// TIA Portal V18 program export: 1 tag tables, 0 data types, 4 data blocks, 6 code blocks (in call order from the OBs), 0 instance data blocks

VAR_GLOBAL   // PLC tag table "AI_Tags"
   AI_Nut_Khoi_Dong AT %I0.0 : Bool;   // Nút khởi động vật lý
   AI_Nut_Khoi_Dong_HMI AT %M110.0 : Bool;   // Tín hiệu mô phỏng/HMI song song cho Nút khởi động vật lý
   AI_Nut_Khoi_Dong_HMI_Gated AT %M320.0 : Bool;   // Tín hiệu HMI đã qua xử lý chế độ cho Nút khởi động vật lý
   AI_Nut_Khoi_Dong_Eff AT %M320.1 : Bool;   // Tín hiệu thực tế/mô phỏng hiệu dụng cho Nút khởi động vật lý
   AI_Nut_Dung AT %I0.1 : Bool;   // Nút dừng vật lý
   AI_Nut_Dung_HMI AT %M110.1 : Bool;   // Tín hiệu mô phỏng/HMI song song cho Nút dừng vật lý
   AI_Nut_Dung_HMI_Gated AT %M320.2 : Bool;   // Tín hiệu HMI đã qua xử lý chế độ cho Nút dừng vật lý
   AI_Nut_Dung_Eff AT %M320.3 : Bool;   // Tín hiệu thực tế/mô phỏng hiệu dụng cho Nút dừng vật lý
   AI_Nut_Reset AT %I0.2 : Bool;   // Nút reset lỗi vật lý
   AI_Nut_Reset_HMI AT %M110.2 : Bool;   // Tín hiệu mô phỏng/HMI song song cho Nút reset lỗi vật lý
   AI_Nut_Reset_HMI_Gated AT %M320.4 : Bool;   // Tín hiệu HMI đã qua xử lý chế độ cho Nút reset lỗi vật lý
   AI_Nut_Reset_Eff AT %M320.5 : Bool;   // Tín hiệu thực tế/mô phỏng hiệu dụng cho Nút reset lỗi vật lý
   AI_Nut_EStop AT %I0.3 : Bool;   // Nút dừng khẩn vật lý
   AI_Nut_EStop_HMI AT %M110.3 : Bool;   // Tín hiệu mô phỏng/HMI song song cho Nút dừng khẩn vật lý
   AI_Nut_EStop_HMI_Gated AT %M320.6 : Bool;   // Tín hiệu HMI đã qua xử lý chế độ cho Nút dừng khẩn vật lý
   AI_Nut_EStop_Eff AT %M320.7 : Bool;   // Tín hiệu thực tế/mô phỏng hiệu dụng cho Nút dừng khẩn vật lý
   AI_FT3200_Bon1 AT %ID100 : Real;   // Cảm biến lưu lượng nước dosing vào Bồn 1
   AI_FT3200_Bon1_HMI AT %MD700 : Real;   // Giá trị mô phỏng/HMI song song cho Cảm biến lưu lượng nước dosing vào Bồn 1
   AI_FT3200_Bon1_Use_HMI AT %M420.0 : Bool;   // Chọn chế độ mô phỏng HMI cho Cảm biến lưu lượng nước dosing vào Bồn 1
   AI_FT3200_Bon1_Sim_Req AT %M321.0 : Bool;   // Yêu cầu mô phỏng cảm biến cho Cảm biến lưu lượng nước dosing vào Bồn 1
   AI_FT3200_Bon1_Sim_Active AT %M321.1 : Bool;   // Mô phỏng cảm biến đang hoạt động cho Cảm biến lưu lượng nước dosing vào Bồn 1
   AI_FT3200_Bon1_Eff AT %MD704 : Real;   // Giá trị thực tế/mô phỏng hiệu dụng cho Cảm biến lưu lượng nước dosing vào Bồn 1
   AI_FQ3200_Bon1 AT %ID104 : Real;   // Bộ đếm lưu lượng tích lũy Bồn 1
   AI_FQ3200_Bon1_HMI AT %MD708 : Real;   // Giá trị mô phỏng/HMI song song cho Bộ đếm lưu lượng tích lũy Bồn 1
   AI_FQ3200_Bon1_Use_HMI AT %M420.1 : Bool;   // Chọn chế độ mô phỏng HMI cho Bộ đếm lưu lượng tích lũy Bồn 1
   AI_FQ3200_Bon1_Sim_Req AT %M321.2 : Bool;   // Yêu cầu mô phỏng cảm biến cho Bộ đếm lưu lượng tích lũy Bồn 1
   AI_FQ3200_Bon1_Sim_Active AT %M321.3 : Bool;   // Mô phỏng cảm biến đang hoạt động cho Bộ đếm lưu lượng tích lũy Bồn 1
   AI_FQ3200_Bon1_Eff AT %MD712 : Real;   // Giá trị thực tế/mô phỏng hiệu dụng cho Bộ đếm lưu lượng tích lũy Bồn 1
   AI_LS3202_Bon1_Cao AT %I0.4 : Bool;   // Cảm biến mức cao Bồn 1
   AI_LS3202_Bon1_Cao_HMI AT %M110.4 : Bool;   // Tín hiệu mô phỏng/HMI song song cho Cảm biến mức cao Bồn 1
   AI_LS3202_Bon1_Cao_HMI_Gated AT %M321.4 : Bool;   // Tín hiệu HMI đã qua xử lý chế độ cho Cảm biến mức cao Bồn 1
   AI_LS3202_Bon1_Cao_Eff AT %M321.5 : Bool;   // Tín hiệu thực tế/mô phỏng hiệu dụng cho Cảm biến mức cao Bồn 1
   AI_LT3203_Bon1 AT %ID108 : Real;   // Cảm biến mức liên tục Bồn 1
   AI_LT3203_Bon1_HMI AT %MD716 : Real;   // Giá trị mô phỏng/HMI song song cho Cảm biến mức liên tục Bồn 1
   AI_LT3203_Bon1_Use_HMI AT %M420.2 : Bool;   // Chọn chế độ mô phỏng HMI cho Cảm biến mức liên tục Bồn 1
   AI_LT3203_Bon1_Sim_Req AT %M321.6 : Bool;   // Yêu cầu mô phỏng cảm biến cho Cảm biến mức liên tục Bồn 1
   AI_LT3203_Bon1_Sim_Active AT %M321.7 : Bool;   // Mô phỏng cảm biến đang hoạt động cho Cảm biến mức liên tục Bồn 1
   AI_LT3203_Bon1_Eff AT %MD720 : Real;   // Giá trị thực tế/mô phỏng hiệu dụng cho Cảm biến mức liên tục Bồn 1
   AI_TT3204_Bon1 AT %ID112 : Real;   // Cảm biến nhiệt độ Bồn 1
   AI_TT3204_Bon1_HMI AT %MD724 : Real;   // Giá trị mô phỏng/HMI song song cho Cảm biến nhiệt độ Bồn 1
   AI_TT3204_Bon1_Use_HMI AT %M420.3 : Bool;   // Chọn chế độ mô phỏng HMI cho Cảm biến nhiệt độ Bồn 1
   AI_TT3204_Bon1_Sim_Req AT %M322.0 : Bool;   // Yêu cầu mô phỏng cảm biến cho Cảm biến nhiệt độ Bồn 1
   AI_TT3204_Bon1_Sim_Active AT %M322.1 : Bool;   // Mô phỏng cảm biến đang hoạt động cho Cảm biến nhiệt độ Bồn 1
   AI_TT3204_Bon1_Eff AT %MD728 : Real;   // Giá trị thực tế/mô phỏng hiệu dụng cho Cảm biến nhiệt độ Bồn 1
   AI_FT3205_Bon2 AT %ID116 : Real;   // Cảm biến lưu lượng nước dosing vào Bồn 2
   AI_FT3205_Bon2_HMI AT %MD732 : Real;   // Giá trị mô phỏng/HMI song song cho Cảm biến lưu lượng nước dosing vào Bồn 2
   AI_FT3205_Bon2_Use_HMI AT %M420.4 : Bool;   // Chọn chế độ mô phỏng HMI cho Cảm biến lưu lượng nước dosing vào Bồn 2
   AI_FT3205_Bon2_Sim_Req AT %M322.2 : Bool;   // Yêu cầu mô phỏng cảm biến cho Cảm biến lưu lượng nước dosing vào Bồn 2
   AI_FT3205_Bon2_Sim_Active AT %M322.3 : Bool;   // Mô phỏng cảm biến đang hoạt động cho Cảm biến lưu lượng nước dosing vào Bồn 2
   AI_FT3205_Bon2_Eff AT %MD736 : Real;   // Giá trị thực tế/mô phỏng hiệu dụng cho Cảm biến lưu lượng nước dosing vào Bồn 2
   AI_FQ3205_Bon2 AT %ID120 : Real;   // Bộ đếm lưu lượng tích lũy Bồn 2
   AI_FQ3205_Bon2_HMI AT %MD740 : Real;   // Giá trị mô phỏng/HMI song song cho Bộ đếm lưu lượng tích lũy Bồn 2
   AI_FQ3205_Bon2_Use_HMI AT %M420.5 : Bool;   // Chọn chế độ mô phỏng HMI cho Bộ đếm lưu lượng tích lũy Bồn 2
   AI_FQ3205_Bon2_Sim_Req AT %M322.4 : Bool;   // Yêu cầu mô phỏng cảm biến cho Bộ đếm lưu lượng tích lũy Bồn 2
   AI_FQ3205_Bon2_Sim_Active AT %M322.5 : Bool;   // Mô phỏng cảm biến đang hoạt động cho Bộ đếm lưu lượng tích lũy Bồn 2
   AI_FQ3205_Bon2_Eff AT %MD744 : Real;   // Giá trị thực tế/mô phỏng hiệu dụng cho Bộ đếm lưu lượng tích lũy Bồn 2
   AI_LT3209_Bon2 AT %ID124 : Real;   // Cảm biến mức liên tục Bồn 2
   AI_LT3209_Bon2_HMI AT %MD748 : Real;   // Giá trị mô phỏng/HMI song song cho Cảm biến mức liên tục Bồn 2
   AI_LT3209_Bon2_Use_HMI AT %M420.6 : Bool;   // Chọn chế độ mô phỏng HMI cho Cảm biến mức liên tục Bồn 2
   AI_LT3209_Bon2_Sim_Req AT %M322.6 : Bool;   // Yêu cầu mô phỏng cảm biến cho Cảm biến mức liên tục Bồn 2
   AI_LT3209_Bon2_Sim_Active AT %M322.7 : Bool;   // Mô phỏng cảm biến đang hoạt động cho Cảm biến mức liên tục Bồn 2
   AI_LT3209_Bon2_Eff AT %MD752 : Real;   // Giá trị thực tế/mô phỏng hiệu dụng cho Cảm biến mức liên tục Bồn 2
   AI_TT3208_Bon2 AT %ID128 : Real;   // Cảm biến nhiệt độ Bồn 2
   AI_TT3208_Bon2_HMI AT %MD756 : Real;   // Giá trị mô phỏng/HMI song song cho Cảm biến nhiệt độ Bồn 2
   AI_TT3208_Bon2_Use_HMI AT %M420.7 : Bool;   // Chọn chế độ mô phỏng HMI cho Cảm biến nhiệt độ Bồn 2
   AI_TT3208_Bon2_Sim_Req AT %M323.0 : Bool;   // Yêu cầu mô phỏng cảm biến cho Cảm biến nhiệt độ Bồn 2
   AI_TT3208_Bon2_Sim_Active AT %M323.1 : Bool;   // Mô phỏng cảm biến đang hoạt động cho Cảm biến nhiệt độ Bồn 2
   AI_TT3208_Bon2_Eff AT %MD760 : Real;   // Giá trị thực tế/mô phỏng hiệu dụng cho Cảm biến nhiệt độ Bồn 2
   AI_V3230_Nuoc_Bon1 AT %Q0.0 : Bool;   // Van on/off cấp nước Bồn 1
   AI_V3230_Nuoc_Bon1_M AT %M220.0 : Bool;   // Tag gương phản hồi HMI cho Van on/off cấp nước Bồn 1
   AI_CV3201_Nuoc_Bon1 AT %QD100 : Real;   // Van tuyến tính cấp nước Bồn 1
   AI_CV3201_Nuoc_Bon1_M AT %MD1200 : Real;   // Tag gương phản hồi HMI cho Van tuyến tính cấp nước Bồn 1
   AI_AGTR3260_Khuay_Bon1 AT %Q0.1 : Bool;   // Động cơ khuấy Bồn 1
   AI_AGTR3260_Khuay_Bon1_M AT %M220.1 : Bool;   // Tag gương phản hồi HMI cho Động cơ khuấy Bồn 1
   AI_AGTR3260_Toc_Do_AO AT %QD104 : Real;   // Tín hiệu tốc độ khuấy Bồn 1
   AI_AGTR3260_Toc_Do_AO_M AT %MD1204 : Real;   // Tag gương phản hồi HMI cho Tín hiệu tốc độ khuấy Bồn 1
   AI_V3232_Xa_Bon1 AT %Q0.2 : Bool;   // Van xả đáy Bồn 1 số 1
   AI_V3232_Xa_Bon1_M AT %M220.2 : Bool;   // Tag gương phản hồi HMI cho Van xả đáy Bồn 1 số 1
   AI_V3233_Xa_Bon1 AT %Q0.3 : Bool;   // Van xả đáy Bồn 1 số 2
   AI_V3233_Xa_Bon1_M AT %M220.3 : Bool;   // Tag gương phản hồi HMI cho Van xả đáy Bồn 1 số 2
   AI_V3234_Xa_Bon1 AT %Q0.4 : Bool;   // Van xả đáy Bồn 1 số 3
   AI_V3234_Xa_Bon1_M AT %M220.4 : Bool;   // Tag gương phản hồi HMI cho Van xả đáy Bồn 1 số 3
   AI_V3235_Nuoc_Bon2 AT %Q0.5 : Bool;   // Van on/off cấp nước Bồn 2
   AI_V3235_Nuoc_Bon2_M AT %M220.5 : Bool;   // Tag gương phản hồi HMI cho Van on/off cấp nước Bồn 2
   AI_CV3206_Hoi_Bon2 AT %QD108 : Real;   // Van hơi/nhiệt Bồn 2 ở chế độ cho phép
   AI_CV3206_Hoi_Bon2_M AT %MD1208 : Real;   // Tag gương phản hồi HMI cho Van hơi/nhiệt Bồn 2 ở chế độ cho phép
   AI_VFD_Bon2_Run AT %Q0.6 : Bool;   // Lệnh chạy VFD động cơ Bồn 2
   AI_VFD_Bon2_Run_M AT %M220.6 : Bool;   // Tag gương phản hồi HMI cho Lệnh chạy VFD động cơ Bồn 2
   AI_VFD_Bon2_Dao_Chieu AT %Q0.7 : Bool;   // Lệnh đảo chiều VFD động cơ Bồn 2
   AI_VFD_Bon2_Dao_Chieu_M AT %M220.7 : Bool;   // Tag gương phản hồi HMI cho Lệnh đảo chiều VFD động cơ Bồn 2
   AI_VFD_Bon2_Toc_Do_AO AT %QD112 : Real;   // Tốc độ đặt VFD Bồn 2 từ HMI setpoint
   AI_VFD_Bon2_Toc_Do_AO_M AT %MD1212 : Real;   // Tag gương phản hồi HMI cho Tốc độ đặt VFD Bồn 2 từ HMI setpoint
   AI_V3237_Xa_Bon2 AT %Q1.0 : Bool;   // Van xả đáy Bồn 2 số 1
   AI_V3237_Xa_Bon2_M AT %M221.0 : Bool;   // Tag gương phản hồi HMI cho Van xả đáy Bồn 2 số 1
   AI_V3238_Xa_Bon2 AT %Q1.1 : Bool;   // Van xả đáy Bồn 2 số 2
   AI_V3238_Xa_Bon2_M AT %M221.1 : Bool;   // Tag gương phản hồi HMI cho Van xả đáy Bồn 2 số 2
   AI_V3239_Xa_Bon2 AT %Q1.2 : Bool;   // Van xả đáy Bồn 2 số 3
   AI_V3239_Xa_Bon2_M AT %M221.2 : Bool;   // Tag gương phản hồi HMI cho Van xả đáy Bồn 2 số 3
   AI_Pump3264_Chuyen_Nhanh1 AT %Q1.3 : Bool;   // Bơm chuyển dung dịch Nhánh 1 xuống bồn chứa
   AI_Pump3264_Chuyen_Nhanh1_M AT %M221.3 : Bool;   // Tag gương phản hồi HMI cho Bơm chuyển dung dịch Nhánh 1 xuống bồn chứa
   AI_LT3302_BonChua1 AT %ID164 : Real;   // Cảm biến mức liên tục Bồn chứa 01
   AI_LT3302_BonChua1_HMI AT %MD828 : Real;   // Giá trị mô phỏng/HMI song song cho Cảm biến mức liên tục Bồn chứa 01
   AI_LT3302_BonChua1_Use_HMI AT %M422.0 : Bool;   // Chọn chế độ mô phỏng HMI cho Cảm biến mức liên tục Bồn chứa 01
   AI_LT3302_BonChua1_Sim_Req AT %M325.4 : Bool;   // Yêu cầu mô phỏng cảm biến cho Cảm biến mức liên tục Bồn chứa 01
   AI_LT3302_BonChua1_Sim_Active AT %M325.5 : Bool;   // Mô phỏng cảm biến đang hoạt động cho Cảm biến mức liên tục Bồn chứa 01
   AI_LT3302_BonChua1_Eff AT %MD832 : Real;   // Giá trị thực tế/mô phỏng hiệu dụng cho Cảm biến mức liên tục Bồn chứa 01
   AI_TT3301_BonChua1 AT %ID168 : Real;   // Cảm biến nhiệt độ Bồn chứa 01
   AI_TT3301_BonChua1_HMI AT %MD836 : Real;   // Giá trị mô phỏng/HMI song song cho Cảm biến nhiệt độ Bồn chứa 01
   AI_TT3301_BonChua1_Use_HMI AT %M422.1 : Bool;   // Chọn chế độ mô phỏng HMI cho Cảm biến nhiệt độ Bồn chứa 01
   AI_TT3301_BonChua1_Sim_Req AT %M325.6 : Bool;   // Yêu cầu mô phỏng cảm biến cho Cảm biến nhiệt độ Bồn chứa 01
   AI_TT3301_BonChua1_Sim_Active AT %M325.7 : Bool;   // Mô phỏng cảm biến đang hoạt động cho Cảm biến nhiệt độ Bồn chứa 01
   AI_TT3301_BonChua1_Eff AT %MD840 : Real;   // Giá trị thực tế/mô phỏng hiệu dụng cho Cảm biến nhiệt độ Bồn chứa 01
   AI_TT3303_TraoDoiNhiet AT %ID172 : Real;   // Cảm biến nhiệt độ bộ trao đổi nhiệt
   AI_TT3303_TraoDoiNhiet_HMI AT %MD844 : Real;   // Giá trị mô phỏng/HMI song song cho Cảm biến nhiệt độ bộ trao đổi nhiệt
   AI_TT3303_TraoDoiNhiet_Use_HMI AT %M422.2 : Bool;   // Chọn chế độ mô phỏng HMI cho Cảm biến nhiệt độ bộ trao đổi nhiệt
   AI_TT3303_TraoDoiNhiet_Sim_Req AT %M326.0 : Bool;   // Yêu cầu mô phỏng cảm biến cho Cảm biến nhiệt độ bộ trao đổi nhiệt
   AI_TT3303_TraoDoiNhiet_Sim_Active AT %M326.1 : Bool;   // Mô phỏng cảm biến đang hoạt động cho Cảm biến nhiệt độ bộ trao đổi nhiệt
   AI_TT3303_TraoDoiNhiet_Eff AT %MD848 : Real;   // Giá trị thực tế/mô phỏng hiệu dụng cho Cảm biến nhiệt độ bộ trao đổi nhiệt
   AI_LT3307_BonChua2 AT %ID176 : Real;   // Cảm biến mức liên tục Bồn chứa 02
   AI_LT3307_BonChua2_HMI AT %MD852 : Real;   // Giá trị mô phỏng/HMI song song cho Cảm biến mức liên tục Bồn chứa 02
   AI_LT3307_BonChua2_Use_HMI AT %M422.3 : Bool;   // Chọn chế độ mô phỏng HMI cho Cảm biến mức liên tục Bồn chứa 02
   AI_LT3307_BonChua2_Sim_Req AT %M326.2 : Bool;   // Yêu cầu mô phỏng cảm biến cho Cảm biến mức liên tục Bồn chứa 02
   AI_LT3307_BonChua2_Sim_Active AT %M326.3 : Bool;   // Mô phỏng cảm biến đang hoạt động cho Cảm biến mức liên tục Bồn chứa 02
   AI_LT3307_BonChua2_Eff AT %MD856 : Real;   // Giá trị thực tế/mô phỏng hiệu dụng cho Cảm biến mức liên tục Bồn chứa 02
   AI_TT3306_BonChua2 AT %ID180 : Real;   // Cảm biến nhiệt độ Bồn chứa 02
   AI_TT3306_BonChua2_HMI AT %MD860 : Real;   // Giá trị mô phỏng/HMI song song cho Cảm biến nhiệt độ Bồn chứa 02
   AI_TT3306_BonChua2_Use_HMI AT %M422.4 : Bool;   // Chọn chế độ mô phỏng HMI cho Cảm biến nhiệt độ Bồn chứa 02
   AI_TT3306_BonChua2_Sim_Req AT %M326.4 : Bool;   // Yêu cầu mô phỏng cảm biến cho Cảm biến nhiệt độ Bồn chứa 02
   AI_TT3306_BonChua2_Sim_Active AT %M326.5 : Bool;   // Mô phỏng cảm biến đang hoạt động cho Cảm biến nhiệt độ Bồn chứa 02
   AI_TT3306_BonChua2_Eff AT %MD864 : Real;   // Giá trị thực tế/mô phỏng hiệu dụng cho Cảm biến nhiệt độ Bồn chứa 02
   AI_PI3308_Truoc_Filter AT %ID184 : Real;   // Cảm biến áp suất trước màng lọc
   AI_PI3308_Truoc_Filter_HMI AT %MD868 : Real;   // Giá trị mô phỏng/HMI song song cho Cảm biến áp suất trước màng lọc
   AI_PI3308_Truoc_Filter_Use_HMI AT %M422.5 : Bool;   // Chọn chế độ mô phỏng HMI cho Cảm biến áp suất trước màng lọc
   AI_PI3308_Truoc_Filter_Sim_Req AT %M326.6 : Bool;   // Yêu cầu mô phỏng cảm biến cho Cảm biến áp suất trước màng lọc
   AI_PI3308_Truoc_Filter_Sim_Active AT %M326.7 : Bool;   // Mô phỏng cảm biến đang hoạt động cho Cảm biến áp suất trước màng lọc
   AI_PI3308_Truoc_Filter_Eff AT %MD872 : Real;   // Giá trị thực tế/mô phỏng hiệu dụng cho Cảm biến áp suất trước màng lọc
   AI_FT3309_Xa_Thanh_Pham AT %ID188 : Real;   // Cảm biến lưu lượng xả thành phẩm
   AI_FT3309_Xa_Thanh_Pham_HMI AT %MD876 : Real;   // Giá trị mô phỏng/HMI song song cho Cảm biến lưu lượng xả thành phẩm
   AI_FT3309_Xa_Thanh_Pham_Use_HMI AT %M422.6 : Bool;   // Chọn chế độ mô phỏng HMI cho Cảm biến lưu lượng xả thành phẩm
   AI_FT3309_Xa_Thanh_Pham_Sim_Req AT %M327.0 : Bool;   // Yêu cầu mô phỏng cảm biến cho Cảm biến lưu lượng xả thành phẩm
   AI_FT3309_Xa_Thanh_Pham_Sim_Active AT %M327.1 : Bool;   // Mô phỏng cảm biến đang hoạt động cho Cảm biến lưu lượng xả thành phẩm
   AI_FT3309_Xa_Thanh_Pham_Eff AT %MD880 : Real;   // Giá trị thực tế/mô phỏng hiệu dụng cho Cảm biến lưu lượng xả thành phẩm
   AI_LSH3310_Pheu_Cao AT %I0.6 : Bool;   // Cảm biến mức cao phễu chiết rót
   AI_LSH3310_Pheu_Cao_HMI AT %M110.6 : Bool;   // Tín hiệu mô phỏng/HMI song song cho Cảm biến mức cao phễu chiết rót
   AI_LSH3310_Pheu_Cao_HMI_Gated AT %M327.2 : Bool;   // Tín hiệu HMI đã qua xử lý chế độ cho Cảm biến mức cao phễu chiết rót
   AI_LSH3310_Pheu_Cao_Eff AT %M327.3 : Bool;   // Tín hiệu thực tế/mô phỏng hiệu dụng cho Cảm biến mức cao phễu chiết rót
   AI_LSL3311_Pheu_Thap AT %I0.7 : Bool;   // Cảm biến mức thấp phễu chiết rót
   AI_LSL3311_Pheu_Thap_HMI AT %M110.7 : Bool;   // Tín hiệu mô phỏng/HMI song song cho Cảm biến mức thấp phễu chiết rót
   AI_LSL3311_Pheu_Thap_HMI_Gated AT %M327.4 : Bool;   // Tín hiệu HMI đã qua xử lý chế độ cho Cảm biến mức thấp phễu chiết rót
   AI_LSL3311_Pheu_Thap_Eff AT %M327.5 : Bool;   // Tín hiệu thực tế/mô phỏng hiệu dụng cho Cảm biến mức thấp phễu chiết rót
   AI_V3331_Xa_BonChua1 AT %Q3.0 : Bool;   // Van xả đáy Bồn chứa 01 số 1
   AI_V3331_Xa_BonChua1_M AT %M223.0 : Bool;   // Tag gương phản hồi HMI cho Van xả đáy Bồn chứa 01 số 1
   AI_V3332_Xa_BonChua1 AT %Q3.1 : Bool;   // Van xả đáy Bồn chứa 01 số 2
   AI_V3332_Xa_BonChua1_M AT %M223.1 : Bool;   // Tag gương phản hồi HMI cho Van xả đáy Bồn chứa 01 số 2
   AI_Pump3361_LuanChuyen_BonChua1 AT %Q3.2 : Bool;   // Bơm luân chuyển Bồn chứa 01
   AI_Pump3361_LuanChuyen_BonChua1_M AT %M223.2 : Bool;   // Tag gương phản hồi HMI cho Bơm luân chuyển Bồn chứa 01
   AI_Pump3362_Xa_BonChua1 AT %Q3.3 : Bool;   // Bơm xả Bồn chứa 01
   AI_Pump3362_Xa_BonChua1_M AT %M223.3 : Bool;   // Tag gương phản hồi HMI cho Bơm xả Bồn chứa 01
   AI_V3333_DieuHuong_BonChua1 AT %Q3.4 : Bool;   // Van điều hướng Bồn chứa 01 số 1
   AI_V3333_DieuHuong_BonChua1_M AT %M223.4 : Bool;   // Tag gương phản hồi HMI cho Van điều hướng Bồn chứa 01 số 1
   AI_V3334_DieuHuong_BonChua1 AT %Q3.5 : Bool;   // Van điều hướng Bồn chứa 01 số 2
   AI_V3334_DieuHuong_BonChua1_M AT %M223.5 : Bool;   // Tag gương phản hồi HMI cho Van điều hướng Bồn chứa 01 số 2
   AI_V3335_DieuHuong_BonChua1 AT %Q3.6 : Bool;   // Van điều hướng Bồn chứa 01 số 3
   AI_V3335_DieuHuong_BonChua1_M AT %M223.6 : Bool;   // Tag gương phản hồi HMI cho Van điều hướng Bồn chứa 01 số 3
   AI_CV3304_Nuoc_Lam_Mat AT %QD132 : Real;   // Van tuyến tính nước làm mát
   AI_CV3304_Nuoc_Lam_Mat_M AT %MD1232 : Real;   // Tag gương phản hồi HMI cho Van tuyến tính nước làm mát
   AI_V3338_Xa_BonChua2 AT %Q3.7 : Bool;   // Van xả đáy Bồn chứa 02 số 1
   AI_V3338_Xa_BonChua2_M AT %M223.7 : Bool;   // Tag gương phản hồi HMI cho Van xả đáy Bồn chứa 02 số 1
   AI_V3339_Xa_BonChua2 AT %Q4.0 : Bool;   // Van xả đáy Bồn chứa 02 số 2
   AI_V3339_Xa_BonChua2_M AT %M224.0 : Bool;   // Tag gương phản hồi HMI cho Van xả đáy Bồn chứa 02 số 2
   AI_Pump3364_Filter AT %Q4.1 : Bool;   // Bơm qua màng lọc CCP số 1
   AI_Pump3364_Filter_M AT %M224.1 : Bool;   // Tag gương phản hồi HMI cho Bơm qua màng lọc CCP số 1
   AI_Pump3365_Filter AT %Q4.2 : Bool;   // Bơm qua màng lọc CCP số 2
   AI_Pump3365_Filter_M AT %M224.2 : Bool;   // Tag gương phản hồi HMI cho Bơm qua màng lọc CCP số 2
   AI_V3340_Duong_Filter AT %Q4.3 : Bool;   // Van đường ống Filter số 1
   AI_V3340_Duong_Filter_M AT %M224.3 : Bool;   // Tag gương phản hồi HMI cho Van đường ống Filter số 1
   AI_V3341_Duong_Filter AT %Q4.4 : Bool;   // Van đường ống Filter số 2
   AI_V3341_Duong_Filter_M AT %M224.4 : Bool;   // Tag gương phản hồi HMI cho Van đường ống Filter số 2
   AI_CV_Filler_Cap_Dich AT %QD136 : Real;   // Van tuyến tính cấp dịch xuống phễu chiết rót
   AI_CV_Filler_Cap_Dich_M AT %MD1236 : Real;   // Tag gương phản hồi HMI cho Van tuyến tính cấp dịch xuống phễu chiết rót
   AI_Coi_Bao_Dong AT %Q4.5 : Bool;   // Còi báo động chung
   AI_Coi_Bao_Dong_M AT %M224.5 : Bool;   // Tag gương phản hồi HMI cho Còi báo động chung
   AI_HMI_Operator_Login AT %M422.7 : Bool;   // Đăng nhập quyền Operator
   AI_HMI_Engineer_Login AT %M423.0 : Bool;   // Đăng nhập quyền Engineer
   AI_HMI_Admin_Login AT %M423.1 : Bool;   // Đăng nhập quyền Admin
   AI_HMI_Che_Do_Manual AT %M423.2 : Bool;   // Cho phép điều khiển tay từng thiết bị
   AI_HMI_Ack_Alarm AT %M423.3 : Bool;   // Xác nhận cảnh báo
   AI_HMI_Reset_Alarm AT %M423.4 : Bool;   // Reset alarm bằng HMI
   AI_Gia_Lap_Mat_Ket_Noi_HMI AT %M423.5 : Bool;   // Nút giả lập mất kết nối PLC
   AI_HMI_User_Level AT %MW520 : Int;   // Mức quyền hiện tại: 1 Operator, 2 Engineer, 3 Admin
   AI_HMI_Cho_Phep_Sua_Thong_So AT %M327.6 : Bool;   // Cờ cho phép sửa công thức và PID
   AI_HMI_Alarm_Status AT %MW522 : Int;   // Mã cảnh báo tổng hợp cho WinCC TextList
   AI_HMI_AnToan_Status AT %MW524 : Int;   // Mã chẩn đoán an toàn ưu tiên
   AI_PLC1_Auto_Enable AT %M327.7 : Bool;   // Cho phép chạy Auto Nhánh 1 Bồn 1-2
   AI_PLC1_EStop_Latch AT %M328.0 : Bool;   // Chốt dừng khẩn HMI/SCADA Nhánh 1 Bồn 1-2
   AI_PLC1_Loi_Tong AT %M328.1 : Bool;   // Lỗi tổng khóa Auto Nhánh 1 Bồn 1-2
   AI_PLC1_Loi_Dry_Run AT %M328.2 : Bool;   // Lỗi chạy khô bơm Nhánh 1 Bồn 1-2
   AI_PLC1_Loi_Dosing AT %M328.3 : Bool;   // Lỗi quá thời gian dosing Nhánh 1 Bồn 1-2
   AI_PLC1_Loi_Truyen_Thong AT %M328.4 : Bool;   // Lỗi truyền thông mô phỏng Nhánh 1 Bồn 1-2
   AI_PLC1_State AT %MW526 : Int;   // Mã bước chu trình Nhánh 1 Bồn 1-2
   AI_PLC1_Step_Bon1_Dosing AT %M329.3 : Bool;   // Bồn 1 đang dosing nước
   AI_PLC1_Step_Bon1_Tip AT %M329.4 : Bool;   // Bồn 1 đang mô phỏng tip cốt tương Nhật Bản
   AI_PLC1_Step_Bon1_Khuay AT %M329.5 : Bool;   // Bồn 1 đang khuấy ban đầu
   AI_PLC1_Step_Bon1_Xa AT %M329.6 : Bool;   // Bồn 1 đang xả sang Bồn 2
   AI_PLC1_Step_Bon2_Dosing AT %M329.7 : Bool;   // Bồn 2 đang dosing bổ sung
   AI_PLC1_Step_Bon2_Tip AT %M330.0 : Bool;   // Bồn 2 đang tip phụ gia
   AI_PLC1_Step_Bon2_Khuay_Thuan AT %M330.1 : Bool;   // Bồn 2 khuấy chiều thuận
   AI_PLC1_Step_Bon2_Khuay_Nghich AT %M330.2 : Bool;   // Bồn 2 khuấy chiều ngược
   AI_PLC1_Step_Bon2_PID AT %M330.3 : Bool;   // Bồn 2 gia nhiệt PID
   AI_PLC1_Step_Bon2_Thanh_Trung AT %M330.4 : Bool;   // Bồn 2 giữ thời gian thanh trùng
   AI_PLC1_Me_Nhanh1_Hoan_Thanh AT %M330.5 : Bool;   // Nhánh 1 hoàn thành và sẵn sàng xả xuống bồn chứa
   AI_PLC1_Xa_Bon1_Xong AT %M330.6 : Bool;   // Bồn 1 đã xả hết
   AI_PLC1_Xa_Bon2_Xong AT %M330.7 : Bool;   // Bồn 2 đã xả hết
   AI_BonChua_Step_Nhan_Dich AT %M332.4 : Bool;   // Bồn chứa 01 đang nhận dịch từ nhánh hoàn thành
   AI_BonChua_Step_Giai_Nhiet AT %M332.5 : Bool;   // Bồn chứa 01 đang giải nhiệt xuống 45 độ C
   AI_BonChua_Step_Chuyen_Bon2 AT %M332.6 : Bool;   // Đang chuyển từ Bồn chứa 01 sang Bồn chứa 02
   AI_BonChua_Step_Loc_Chiet AT %M332.7 : Bool;   // Đang lọc CCP và chiết rót
   AI_BonChua_Me_Hoan_Thanh AT %M333.0 : Bool;   // Hoàn thành một mẻ sản xuất chung
   AI_BonChua_State AT %MW530 : Int;   // Mã bước cụm bồn chứa và lọc thành phẩm
   AI_BonChua_Owner_Nhanh1 AT %M333.1 : Bool;   // Mức ưu tiên Nhánh 1 sở hữu bồn chứa
   AI_BonChua_Owner_Nhanh2 AT %M333.2 : Bool;   // Mức ưu tiên Nhánh 2 sở hữu bồn chứa
   AI_PLC2_Me_Nhanh2_Hoan_Thanh_Nhan AT %M333.4 : Bool;   // Cờ PLC1 nhận trạng thái hoàn thành từ PLC2
   AI_PLC2_Me_Nhanh2_Hoan_Thanh_Nhan_HMI AT %M111.0 : Bool;   // Tín hiệu mô phỏng/HMI song song cho cờ PLC1 nhận trạng thái hoàn thành từ PLC2
   AI_PLC2_Xa_Bon4_Xong_Nhan AT %M333.5 : Bool;   // Cờ PLC1 nhận trạng thái xả xong Bồn 4 từ PLC2
   AI_Pump3265_Chuyen_Nhanh2_Cmd AT %M333.6 : Bool;   // Lệnh chạy bơm chuyển Nhánh 2 gửi sang PLC2
   AI_Pump3265_Chuyen_Nhanh2_Cmd_M AT %M224.7 : Bool;   // Tag gương phản hồi HMI cho lệnh chạy bơm chuyển Nhánh 2 gửi sang PLC2
   AI_PID_Bon4_SP_Recv AT %MD884 : Real;   // PID Bồn 4 Setpoint nhận từ PLC2
   AI_PID_Bon4_PV_Recv AT %MD888 : Real;   // PID Bồn 4 Process Value nhận từ PLC2
   AI_PID_Bon4_CV_Recv AT %MD892 : Real;   // PID Bồn 4 Control Value nhận từ PLC2
   AI_PLC2_State_Recv AT %MW532 : Int;   // Trạng thái hoạt động PLC2 nhận từ PLC2
   AI_PLC2_Loi_Tong_Recv AT %M334.0 : Bool;   // Cờ lỗi tổng PLC2 nhận từ PLC2
   AI_VFD_Bon2_iStep AT %MW60 : Int;   // Bước quét tuần tự Modbus VFD Bồn 2
   AI_VFD_Bon2_iStep_Reset AT %M335.5 : Bool;   // Cờ reset bộ đếm bước Modbus VFD Bồn 2
   AI_VFD_Bon2_Step0_Req AT %M335.6 : Bool;   // Yêu cầu bước 0 Modbus VFD Bồn 2
   AI_VFD_Bon2_Step1_Req AT %M335.7 : Bool;   // Yêu cầu bước 1 Modbus VFD Bồn 2
   AI_VFD_Bon2_Step2_Req AT %M336.0 : Bool;   // Yêu cầu bước 2 Modbus VFD Bồn 2
   AI_VFD_Bon2_Step3_Req AT %M336.1 : Bool;   // Yêu cầu bước 3 Modbus VFD Bồn 2
   AI_VFD_Bon2_MB_ControlWord AT %MW40 : Word;   // Control Word gửi VFD Bồn 2
   AI_VFD_Bon2_MB_FreqSetpoint AT %MW42 : Int;   // Frequency Setpoint gửi VFD Bồn 2
   AI_VFD_Bon2_MB_StatusWord AT %MW44 : Word;   // Status Word đọc từ VFD Bồn 2
   AI_VFD_Bon2_MB_ActualSpeed AT %MW46 : Int;   // Actual Speed đọc từ VFD Bồn 2
   AI_VFD_Bon2_MB_Error AT %M50.0 : Bool;   // Lỗi Modbus Master VFD Bồn 2
   AI_VFD_Bon2_MB_Busy AT %M50.1 : Bool;   // Modbus Master Busy VFD Bồn 2
   AI_VFD_Bon2_MB_Done AT %M50.2 : Bool;   // Modbus Master Done VFD Bồn 2
   AI_VFD_Bon2_MB_Status AT %MW52 : Word;   // Trạng thái Modbus Master VFD Bồn 2
   AI_VFD_Bon2_MBCL_Done AT %M51.0 : Bool;   // Modbus Comm Load Done VFD Bồn 2
   AI_VFD_Bon2_MBCL_Error AT %M51.1 : Bool;   // Modbus Comm Load Error VFD Bồn 2
   AI_VFD_Bon2_MBCL_Status AT %MW54 : Word;   // Trạng thái Modbus Comm Load VFD Bồn 2
   AI_VFD_Bon2_Freq_Temp AT %MD70 : Real;   // Biến tạm tần số VFD Bồn 2
   AI_VFD_Bon2_Actual_Speed_Feedback AT %MD74 : Real;   // Phản hồi tốc độ thực tế VFD Bồn 2
   AI_VFD_Bon2_Actual_Speed_Feedback_M AT %MD1240 : Real;   // Tag gương phản hồi HMI tốc độ thực tế VFD Bồn 2
   AI_Clock_1Hz AT %M100.5 : Bool;   // Clock 1Hz system memory bit
   AI_FirstScan AT %M101.0 : Bool;   // First Scan system memory bit
   AI_MB_TCP_iStep AT %MW80 : Int;   // Modbus TCP Client step
   AI_MB_TCP_REQ AT %M82.0 : Bool;   // Modbus TCP Client Request
   AI_MB_TCP_DONE AT %M82.2 : Bool;   // Modbus TCP Client Transaction Done
   AI_MB_TCP_ERROR AT %M82.3 : Bool;   // Modbus TCP Client Transaction Error
   AI_MB_TCP_BUSY AT %M82.6 : Bool;   // Modbus TCP Client Transaction Busy
   AI_MB_TCP_STATUS AT %MW84 : Word;   // Modbus TCP Client Status
   AI_MB_TCP_Mode AT %MB88 : USInt;   // Modbus TCP Client Mode
   AI_MB_TCP_DataAddr AT %MD90 : UDInt;   // Modbus TCP Client Data Address
   AI_MB_TCP_DataLen AT %MW94 : UInt;   // Modbus TCP Client Data Length
   AI_Nut_Khoi_Dong_Eff_Old AT %M83.0 : Bool;   // Old value of Start button
   AI_Nut_Khoi_Dong_Eff_Edge AT %M83.6 : Bool;   // Start command edge detected
   AI_Nut_Dung_Eff_Old AT %M83.1 : Bool;   // Old value of Stop button
   AI_Nut_Dung_Eff_Edge AT %M83.7 : Bool;   // Stop command edge detected
   AI_Nut_Reset_Eff_Old AT %M83.2 : Bool;   // Old value of Reset button
   AI_Nut_Reset_Eff_Edge AT %M84.0 : Bool;   // Reset command edge detected
   AI_Nut_EStop_Eff_Old AT %M83.3 : Bool;   // Old value of EStop button
   AI_Nut_EStop_Eff_Edge AT %M84.1 : Bool;   // EStop command edge detected
   AI_Pump3265_Chuyen_Nhanh2_Cmd_Old AT %M83.4 : Bool;   // Old value of Transfer command
   AI_Pump3265_Chuyen_Nhanh2_Cmd_Edge AT %M84.2 : Bool;   // Transfer command edge detected
   AI_PLC1_Load_Default_Cmd_Old AT %M83.5 : Bool;   // Old value of Load Recipe command
   AI_PLC1_Load_Default_Cmd_Edge AT %M84.3 : Bool;   // Load Recipe command edge detected
   AI_MB_TCP_Any_Cmd_Edge AT %M84.4 : Bool;   // Any handshake command edge detected
   AI_PLC1_Tip_Bon1_Xong_HMI AT %M423.6 : Bool;   // Nút mô phỏng tip Bồn 1 đã hoàn tất
   AI_PLC1_Khuay_Bon1_Xong_HMI AT %M423.7 : Bool;   // Nút mô phỏng hết thời gian khuấy Bồn 1
   AI_PLC1_Tip_Bon2_Xong_HMI AT %M424.0 : Bool;   // Nút mô phỏng tip Bồn 2 đã hoàn tất
   AI_PLC1_Khuay_Thuan_Bon2_Xong_HMI AT %M424.1 : Bool;   // Nút mô phỏng hết thời gian khuấy thuận Bồn 2
   AI_PLC1_Khuay_Nghich_Bon2_Xong_HMI AT %M424.2 : Bool;   // Nút mô phỏng hết thời gian khuấy ngược Bồn 2
   AI_PLC1_Thanh_Trung_Bon2_Xong_HMI AT %M424.3 : Bool;   // Nút mô phỏng hết thời gian thanh trùng Bồn 2
   AI_PLC2_Tip_Bon3_Xong_HMI AT %M424.4 : Bool;   // Nút mô phỏng tip Bồn 3 đã hoàn tất
   AI_PLC2_Khuay_Bon3_Xong_HMI AT %M424.5 : Bool;   // Nút mô phỏng hết thời gian khuấy Bồn 3
   AI_PLC2_Tip_Bon4_Xong_HMI AT %M424.6 : Bool;   // Nút mô phỏng tip Bồn 4 đã hoàn tất
   AI_PLC2_Khuay_Thuan_Bon4_Xong_HMI AT %M424.7 : Bool;   // Nút mô phỏng hết thời gian khuấy thuận Bồn 4
   AI_PLC2_Khuay_Nghich_Bon4_Xong_HMI AT %M425.0 : Bool;   // Nút mô phỏng hết thời gian khuấy ngược Bồn 4
   AI_PLC2_Thanh_Trung_Bon4_Xong_HMI AT %M425.1 : Bool;   // Nút mô phỏng hết thời gian thanh trùng Bồn 4
   AI_BonChua_Nhan_Dich_Xong_HMI AT %M425.2 : Bool;   // Nút mô phỏng nhận dịch vào Bồn chứa 01 xong
   AI_BonChua_Chuyen_Bon2_Xong_HMI AT %M425.3 : Bool;   // Nút mô phỏng chuyển sang Bồn chứa 02 xong
   AI_HMI_SP_PLC1_Nuoc_Bon1 AT %MD896 : Real;   // Lượng nước dosing Bồn 1
   AI_HMI_SP_PLC1_Nuoc_Bon2 AT %MD900 : Real;   // Lượng nước dosing bổ sung Bồn 2
   AI_HMI_SP_PLC1_Toc_Do_Bon1 AT %MD904 : Real;   // Tốc độ khuấy Bồn 1
   AI_HMI_SP_PLC1_Toc_Do_Bon2_Main AT %MD908 : Real;   // Tốc độ khuấy chính Bồn 2
   AI_HMI_SP_PLC1_Nhiet_Do_Bon2 AT %MD912 : Real;   // Setpoint nhiệt/PID Bồn 2
   AI_HMI_SP_PLC2_Nuoc_Bon3 AT %MD916 : Real;   // Lượng nước dosing Bồn 3
   AI_HMI_SP_PLC2_Nuoc_Bon4 AT %MD920 : Real;   // Lượng nước dosing bổ sung Bồn 4
   AI_HMI_SP_PLC2_Toc_Do_Bon3 AT %MD924 : Real;   // Tốc độ khuấy Bồn 3
   AI_HMI_SP_PLC2_Toc_Do_Bon4_Main AT %MD928 : Real;   // Tốc độ khuấy chính Bồn 4
   AI_HMI_SP_PLC2_Nhiet_Do_Bon4 AT %MD932 : Real;   // Setpoint nhiệt/PID mô phỏng Bồn 4
   AI_HMI_SP_BonChua1_Nhiet_Giai_Nhiet AT %MD936 : Real;   // Nhiệt độ giải nhiệt đích Bồn chứa 01
   AI_HMI_SP_Loc_Ap_Suat_Max AT %MD940 : Real;   // Ngưỡng áp suất cao trước màng lọc
   AI_HMI_SP_Time_Khuay_Bon1 AT %MD944 : Time;   // Thời gian khuấy Bồn 1
   AI_HMI_SP_Time_Khuay_Bon3 AT %MD948 : Time;   // Thời gian khuấy Bồn 3
   AI_HMI_SP_Time_Fwd AT %MD952 : Time;   // Thời gian khuấy chiều thuận
   AI_HMI_SP_Time_Rev AT %MD956 : Time;   // Thời gian khuấy chiều ngược
   AI_HMI_SP_Time_Sterilize AT %MD960 : Time;   // Thời gian giữ nhiệt thanh trùng
   AI_PLC1_Khuay_Bon1_Xong AT %M336.2 : Bool;   // Trạng thái tự động xong khuấy Bồn 1
   AI_PLC1_Khuay_Thuan_Bon2_Xong AT %M336.3 : Bool;   // Trạng thái tự động xong khuấy thuận Bồn 2
   AI_PLC1_Khuay_Nghich_Bon2_Xong AT %M336.4 : Bool;   // Trạng thái tự động xong khuấy ngược Bồn 2
   AI_PLC1_Thanh_Trung_Bon2_Xong AT %M336.5 : Bool;   // Trạng thái tự động xong thanh trùng Bồn 2
   AI_PLC2_Khuay_Bon3_Xong AT %M336.6 : Bool;   // Trạng thái tự động xong khuấy Bồn 3
   AI_PLC2_Khuay_Thuan_Bon4_Xong AT %M336.7 : Bool;   // Trạng thái tự động xong khuấy thuận Bồn 4
   AI_PLC2_Khuay_Nghich_Bon4_Xong AT %M337.0 : Bool;   // Trạng thái tự động xong khuấy ngược Bồn 4
   AI_PLC2_Thanh_Trung_Bon4_Xong AT %M337.1 : Bool;   // Trạng thái tự động xong thanh trùng Bồn 4
   AI_PLC1_Tip_Bon1_Auto_Done AT %M337.2 : Bool;   // Trạng thái tự động xong tip Bồn 1
   AI_PLC1_Tip_Bon2_Auto_Done AT %M337.3 : Bool;   // Trạng thái tự động xong tip Bồn 2
   AI_PLC2_Tip_Bon3_Auto_Done AT %M337.4 : Bool;   // Trạng thái tự động xong tip Bồn 3
   AI_PLC2_Tip_Bon4_Auto_Done AT %M337.5 : Bool;   // Trạng thái tự động xong tip Bồn 4
   AI_PLC1_Start_Edge_Old AT %M337.6 : Bool;   // Cờ nhớ cạnh lên nút Start PLC1
   AI_PLC1_Start_Edge_Edge AT %M337.7 : Bool;   // Xung cạnh lên nút Start PLC1
   AI_PLC2_Start_Edge_Old AT %M338.0 : Bool;   // Cờ nhớ cạnh lên nút Start PLC2
   AI_PLC2_Start_Edge_Edge AT %M338.1 : Bool;   // Xung cạnh lên nút Start PLC2
   AI_PID_Bon2_Enable AT %M338.2 : Bool;   // Cho phép PID Bồn 2
   AI_PID_Bon2_ManualEnable AT %M338.3 : Bool;   // Chế độ manual PID Bồn 2
   AI_PID_Bon2_Error AT %M338.4 : Bool;   // Lỗi khối PID Bồn 2
   AI_PID_Bon2_Reset_Eff AT %M338.5 : Bool;   // Reset hiệu dụng PID Bồn 2
   AI_PID_Bon4_Enable AT %M338.6 : Bool;   // Cho phép PID mô phỏng Bồn 4
   AI_PID_Bon4_ManualEnable AT %M338.7 : Bool;   // Chế độ manual PID Bồn 4
   AI_PID_Bon4_Error AT %M339.0 : Bool;   // Lỗi khối PID Bồn 4
   AI_PID_Bon4_Reset_Eff AT %M339.1 : Bool;   // Reset hiệu dụng PID Bồn 4
   AI_PID_Bon2_ErrorBits AT %MD964 : DWord;   // Mã lỗi DWORD PID Bồn 2
   AI_PID_Bon4_ErrorBits AT %MD968 : DWord;   // Mã lỗi DWORD PID Bồn 4
   AI_PID_Bon2_SP AT %MD972 : Real;   // Setpoint đưa vào PID Bồn 2
   AI_PID_Bon2_Err AT %MD976 : Real;   // Sai lệch PID Bồn 2 = SP - PV
   AI_PID_Bon2_CV AT %MD980 : Real;   // Giá trị điều khiển PID Bồn 2
   AI_PID_Bon2_ManualValue AT %MD984 : Real;   // Giá trị manual PID Bồn 2
   AI_PID_Bon4_SP AT %MD988 : Real;   // Setpoint đưa vào PID mô phỏng Bồn 4
   AI_PID_Bon4_Err AT %MD992 : Real;   // Sai lệch PID mô phỏng Bồn 4 = SP - PV
   AI_PID_Bon4_CV AT %MD996 : Real;   // Giá trị điều khiển PID mô phỏng Bồn 4
   AI_PID_Bon4_ManualValue AT %MD1000 : Real;   // Giá trị manual PID Bồn 4
   AI_TT3219_Bon4_Sim AT %MD1004 : Real;   // Nhiệt độ mô phỏng nội bộ cho PID Bồn 4
   AI_PID_Bon2_Temp_Inc AT %MD1008 : Real;   // Mức tăng nhiệt mô phỏng Bồn 2
   AI_PID_Bon4_Tang_Nhiet_Buoc AT %MD1012 : Real;   // Mức tăng nhiệt mô phỏng mỗi chu kỳ OB31
   AI_TT3219_Bon4_Target AT %MD1016 : Real;   // Nhiệt độ đích mô phỏng bồn 4
   AI_TT3219_Bon4_Sim_Pure AT %MD1020 : Real;   // Nhiệt độ mô phỏng chưa có nhiễu bồn 4
   AI_PID_Bon4_Temp_Val_1 AT %MD1024 : Real;   // Biến tạm mô phỏng nhiệt độ 1
   AI_PID_Bon4_Temp_Val_2 AT %MD1028 : Real;   // Biến tạm mô phỏng nhiệt độ 2
   AI_PID_Bon4_Sim_Counter AT %MD1032 : Real;   // Đồng hồ chu kỳ mô phỏng
   AI_PID_Bon4_Sim_Angle AT %MD1036 : Real;   // Góc lượng giác nhiễu
   AI_PID_Bon4_Sim_Sin AT %MD1040 : Real;   // Giá trị hình sin nhiễu
   AI_PID_Bon4_Sim_Noise AT %MD1044 : Real;   // Giá trị nhiễu nhiệt độ
   AI_PLC1_Tip_Bon1_Timer AT %MD1048 : Real;   // Bộ đếm thời gian mô phỏng tip bồn 1
   AI_PLC1_Tip_Bon2_Timer AT %MD1052 : Real;   // Bộ đếm thời gian mô phỏng tip bồn 2
   AI_PLC2_Tip_Bon3_Timer AT %MD1056 : Real;   // Bộ đếm thời gian mô phỏng tip bồn 3
   AI_PLC2_Tip_Bon4_Timer AT %MD1060 : Real;   // Bộ đếm thời gian mô phỏng tip bồn 4
   AI_PID_Bon2_State AT %MW534 : Int;   // Trạng thái khối PID Bồn 2
   AI_PLC1_Stop_Active AT %M339.2 : Bool;   // Tín hiệu dừng active PLC1
   AI_VFD_Bon2_Khuay_Active AT %M339.4 : Bool;   // Trạng thái khuấy Bồn 2 active
   AI_VFD_Bon2_Should_Run AT %M339.5 : Bool;   // Yêu cầu chạy VFD Bồn 2
   AI_HMI_Use_Sim_Input_PLC1 AT %M340.0 : Bool;   // Cho phép sử dụng đầu vào mô phỏng PLC1
   AI_HMI_Use_Sim_Input_BonChua AT %M340.2 : Bool;   // Cho phép sử dụng đầu vào mô phỏng Bồn chứa
   AI_PLC2_Me_Nhanh2_Hoan_Thanh_Nhan_Eff AT %M340.3 : Bool;   // Cờ nhận trạng thái hoàn thành Nhánh 2 hiệu dụng
   AI_PLC2_Me_Nhanh2_Hoan_Thanh_Nhan_HMI_Gated AT %M340.5 : Bool;   // Cờ nhận trạng thái hoàn thành Nhánh 2 HMI gated
   AI_PLC1_SP_Valid AT %M340.7 : Bool;   // Setpoint PLC1 hợp lệ
   AI_BonChua_SP_Valid AT %M341.1 : Bool;   // Setpoint Bồn chứa hợp lệ
   AI_PLC1_Loi_Setpoint AT %M341.2 : Bool;   // Lỗi Setpoint PLC1
   AI_BonChua_Loi_Setpoint AT %M341.4 : Bool;   // Lỗi Setpoint Bồn chứa
   AI_Init_Defaults_Done_PLC1 AT %M341.5 : Bool;   // Khởi tạo Setpoint mặc định PLC1 hoàn tất
   AI_Init_Defaults_Done_BonChua AT %M341.7 : Bool;   // Khởi tạo Setpoint mặc định Bồn chứa hoàn tất
   AI_Init_Trigger_PLC1 AT %M342.0 : Bool;   // Cờ kích hoạt nạp recipe mặc định PLC1
   AI_Init_Trigger_BonChua AT %M342.2 : Bool;   // Cờ kích hoạt nạp recipe mặc định Bồn chứa
   AI_HMI_Load_Default_Recipe AT %M342.3 : Bool;   // Yêu cầu nạp lại Recipe mặc định từ HMI
   AI_PLC1_Load_Default_Cmd AT %M342.4 : Bool;   // Lệnh nạp recipe mặc định gửi sang PLC2
   AI_PLC1_Load_Default_Cmd_M AT %M225.0 : Bool;   // Tag gương phản hồi HMI cho lệnh nạp recipe mặc định PLC1
   AI_PLC1_Load_Default_Done_Nhan AT %M343.1 : Bool;   // Nhận báo nạp recipe xong từ PLC2
   AI_PLC1_Load_Default_Done_Nhan_HMI AT %M111.7 : Bool;   // Tín hiệu mô phỏng/HMI cho nhận báo nạp recipe xong
   AI_PLC1_Load_Default_Done_Nhan_HMI_Gated AT %M343.2 : Bool;   // Tín hiệu nhận báo nạp recipe xong HMI gated
   AI_PLC1_Load_Default_Done_Nhan_Eff AT %M343.3 : Bool;   // Tín hiệu nhận báo nạp recipe xong hiệu dụng
   AI_HMI_Sim_Mode AT %M343.4 : Bool;   // Cho phép toàn bộ tín hiệu mô phỏng HMI tác động vào input hiệu dụng
   AI_HMI_Run_Enable AT %M343.5 : Bool;   // Cho phép vận hành từ HMI ở chế độ thật
   AI_System_Mode_Real AT %M343.6 : Bool;   // Hệ thống đang hoạt động ở chế độ thực tế
   AI_System_Mode_Sim AT %M343.7 : Bool;   // Hệ thống đang hoạt động ở chế độ mô phỏng
   AI_HMI_Sim_Active_Warning AT %M344.0 : Bool;   // Cảnh báo chế độ mô phỏng HMI đang hoạt động
   AI_PID_Bon2_Kp_HMI AT %MD1064 : Real;   // HMI parameter for Kp PID Bồn 2
   AI_PID_Bon2_Ti_HMI AT %MD1068 : Real;   // HMI parameter for Ti PID Bồn 2
   AI_BonChua_Nhan_Dich_Xong_Nhanh1 AT %M344.1 : Bool;   // Nhận dịch xong từ Nhánh 1
   AI_BonChua_Nhan_Dich_Xong_Nhanh2 AT %M344.2 : Bool;   // Nhận dịch xong từ Nhánh 2
   AI_Clock_1Hz_Last AT %M344.3 : Bool;   // Trạng thái Clock 1Hz chu kỳ trước
   AI_Clock_1Hz_Edge AT %M344.4 : Bool;   // Xung cạnh lên của Clock 1Hz
   AI_PLC2_Heartbeat_Last AT %MW540 : Int;   // Heartbeat PLC2 chu kỳ trước
   AI_PLC2_Heartbeat_Changed AT %M344.7 : Bool;   // Cờ heartbeat PLC2 thay đổi
   AI_PLC1_Heartbeat_Timeout AT %M345.0 : Bool;   // Lỗi timeout heartbeat PLC2
   AI_VFD_Bon2_MB_Req AT %M345.1 : Bool;   // REQ cho VFD Modbus
   AI_VFD_Bon2_MB_Mode AT %MB500 : USInt;   // MODE cho VFD Modbus
   AI_VFD_Bon2_MB_DataAddr AT %MD504 : UDInt;   // DATA_ADDR cho VFD Modbus
   AI_VFD_Bon2_MB_DataLen AT %MW508 : UInt;   // DATA_LEN cho VFD Modbus
   AI_VFD_Bon2_MB_DataBuffer AT %MW510 : Word;   // Buffer dữ liệu cho VFD Modbus
END_VAR

DATA_BLOCK "AI_Timers_PLC1"   // DB
TITLE = AI_Timers_PLC1
{ S7_Optimized_Access := 'TRUE' }
VERSION : 0.1
// Global DB containing all timers and PID instances
// stored: AutoNumber true, IsOnlyStoredInLoadMemory false, IsWriteProtectedInAS false
   VAR
      AI_Timer_Dosing_Bon1 : IEC_TIMER;
      AI_Timer_Tip_Bon1 : IEC_TIMER;
      AI_Timer_Dosing_Bon2 : IEC_TIMER;
      AI_Timer_Tip_Bon2 : IEC_TIMER;
      AI_Timer_Khuay_Bon1 : IEC_TIMER;
      AI_Timer_Khuay_Thuan_Bon2 : IEC_TIMER;
      AI_Timer_Khuay_Nghich_Bon2 : IEC_TIMER;
      AI_Timer_Thanh_Trung_Bon2 : IEC_TIMER;
      AI_Timer_DryRun_Bon2 : IEC_TIMER;
      AI_Timer_Heartbeat_PLC1 : IEC_TIMER;
      AI_VFD_Bon2_MB_Counter : IEC_COUNTER;
   END_VAR
BEGIN
END_DATA_BLOCK

DATA_BLOCK "DB_PLC1_MB_Buffer_DB"   // DB12
TITLE = DB_PLC1_MB_Buffer_DB
{ S7_Optimized_Access := 'FALSE' }
VERSION : 0.1
// DB communication via Modbus TCP
// stored: AutoNumber false, IsOnlyStoredInLoadMemory false, IsWriteProtectedInAS false
   VAR
      Send_CmdSeq : Int;
      Send_Cmd_Start : Bool;
      Send_Cmd_Stop : Bool;
      Send_Cmd_Reset : Bool;
      Send_Cmd_EStop : Bool;
      Send_Cmd_Pump_Branch2_To_SubTanks : Bool;
      Send_Cmd_Load_Recipe : Bool;
      Send_Heartbeat : Int;
      Recv_AckSeq : Int;
      Recv_Done_Branch2 : Bool;
      Recv_Done_Recipe : Bool;
      Recv_Alarm : Bool;
      Recv_State : Int;
      Recv_PID_Bon4_SP : Real;
      Recv_PID_Bon4_PV : Real;
      Recv_PID_Bon4_CV : Real;
      Recv_Done_Discharge2 : Bool;
      Recv_Heartbeat : Int;
   END_VAR
BEGIN
END_DATA_BLOCK

DATA_BLOCK "DB_PLC1_Recv_From_PLC2_DB"   // DB10
TITLE = DB_PLC1_Recv_From_PLC2_DB
{ S7_Optimized_Access := 'FALSE' }
VERSION : 0.1
// DB communication via Modbus TCP
// stored: AutoNumber false, IsOnlyStoredInLoadMemory false, IsWriteProtectedInAS false
   VAR
      AckSeq : Int;
      Done_Branch2 : Bool;
      Done_Recipe : Bool;
      Alarm : Bool;
      State : Int;
      PID_Bon4_SP : Real;
      PID_Bon4_PV : Real;
      PID_Bon4_CV : Real;
      Done_Discharge2 : Bool;
      Heartbeat : Int;
   END_VAR
BEGIN
END_DATA_BLOCK

DATA_BLOCK "DB_PLC1_Send_To_PLC2_DB"   // DB11
TITLE = DB_PLC1_Send_To_PLC2_DB
{ S7_Optimized_Access := 'FALSE' }
VERSION : 0.1
// DB communication via Modbus TCP
// stored: AutoNumber false, IsOnlyStoredInLoadMemory false, IsWriteProtectedInAS false
   VAR
      CmdSeq : Int;
      Cmd_Start : Bool;
      Cmd_Stop : Bool;
      Cmd_Reset : Bool;
      Cmd_EStop : Bool;
      Cmd_Pump_Branch2_To_SubTanks : Bool;
      Cmd_Load_Recipe : Bool;
      Heartbeat : Int;
   END_VAR
BEGIN
END_DATA_BLOCK

ORGANIZATION_BLOCK "Main"   // OB1, LAD, ProgramCycle
{ S7_Optimized_Access := 'TRUE' }
VERSION : 0.1
// stored: AutoNumber true, IsIECCheckEnabled false
   VAR_INPUT
      Initial_Call : Bool;
      Remanence : Bool;
   END_VAR
BEGIN

REGION Network 1: Clock 1Hz Edge Detection
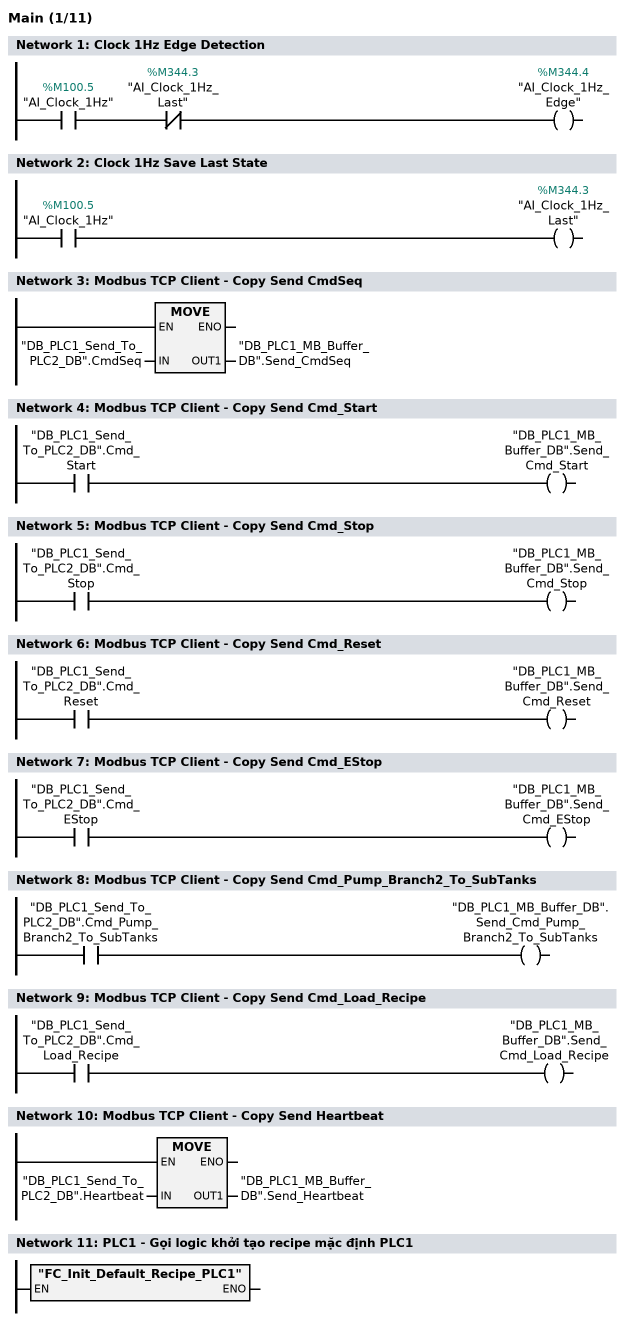
   RUNG wire#powerrail
      Contact( "AI_Clock_1Hz" )
      I_Contact( "AI_Clock_1Hz_Last" )
      Coil( "AI_Clock_1Hz_Edge" )
   END_RUNG
   // the same network as SCL:
   "AI_Clock_1Hz_Edge" := "AI_Clock_1Hz" AND NOT "AI_Clock_1Hz_Last";
END_REGION

REGION Network 2: Clock 1Hz Save Last State
   RUNG wire#powerrail
      Contact( "AI_Clock_1Hz" )
      Coil( "AI_Clock_1Hz_Last" )
   END_RUNG
   // the same network as SCL:
   "AI_Clock_1Hz_Last" := "AI_Clock_1Hz";
END_REGION

REGION Network 3: Modbus TCP Client - Copy Send CmdSeq
   RUNG wire#powerrail
      { S7_GenerateENO := "TRUE" } Move(in := "DB_PLC1_Send_To_PLC2_DB".CmdSeq, out1 => "DB_PLC1_MB_Buffer_DB".Send_CmdSeq)
   END_RUNG
   // the same network as SCL:
   "DB_PLC1_MB_Buffer_DB".Send_CmdSeq := "DB_PLC1_Send_To_PLC2_DB".CmdSeq;
END_REGION

REGION Network 4: Modbus TCP Client - Copy Send Cmd_Start
   RUNG wire#powerrail
      Contact( "DB_PLC1_Send_To_PLC2_DB".Cmd_Start )
      Coil( "DB_PLC1_MB_Buffer_DB".Send_Cmd_Start )
   END_RUNG
   // the same network as SCL:
   "DB_PLC1_MB_Buffer_DB".Send_Cmd_Start := "DB_PLC1_Send_To_PLC2_DB".Cmd_Start;
END_REGION

REGION Network 5: Modbus TCP Client - Copy Send Cmd_Stop
   RUNG wire#powerrail
      Contact( "DB_PLC1_Send_To_PLC2_DB".Cmd_Stop )
      Coil( "DB_PLC1_MB_Buffer_DB".Send_Cmd_Stop )
   END_RUNG
   // the same network as SCL:
   "DB_PLC1_MB_Buffer_DB".Send_Cmd_Stop := "DB_PLC1_Send_To_PLC2_DB".Cmd_Stop;
END_REGION

REGION Network 6: Modbus TCP Client - Copy Send Cmd_Reset
   RUNG wire#powerrail
      Contact( "DB_PLC1_Send_To_PLC2_DB".Cmd_Reset )
      Coil( "DB_PLC1_MB_Buffer_DB".Send_Cmd_Reset )
   END_RUNG
   // the same network as SCL:
   "DB_PLC1_MB_Buffer_DB".Send_Cmd_Reset := "DB_PLC1_Send_To_PLC2_DB".Cmd_Reset;
END_REGION

REGION Network 7: Modbus TCP Client - Copy Send Cmd_EStop
   RUNG wire#powerrail
      Contact( "DB_PLC1_Send_To_PLC2_DB".Cmd_EStop )
      Coil( "DB_PLC1_MB_Buffer_DB".Send_Cmd_EStop )
   END_RUNG
   // the same network as SCL:
   "DB_PLC1_MB_Buffer_DB".Send_Cmd_EStop := "DB_PLC1_Send_To_PLC2_DB".Cmd_EStop;
END_REGION

REGION Network 8: Modbus TCP Client - Copy Send Cmd_Pump_Branch2_To_SubTanks
   RUNG wire#powerrail
      Contact( "DB_PLC1_Send_To_PLC2_DB".Cmd_Pump_Branch2_To_SubTanks )
      Coil( "DB_PLC1_MB_Buffer_DB".Send_Cmd_Pump_Branch2_To_SubTanks )
   END_RUNG
   // the same network as SCL:
   "DB_PLC1_MB_Buffer_DB".Send_Cmd_Pump_Branch2_To_SubTanks := "DB_PLC1_Send_To_PLC2_DB".Cmd_Pump_Branch2_To_SubTanks;
END_REGION

REGION Network 9: Modbus TCP Client - Copy Send Cmd_Load_Recipe
   RUNG wire#powerrail
      Contact( "DB_PLC1_Send_To_PLC2_DB".Cmd_Load_Recipe )
      Coil( "DB_PLC1_MB_Buffer_DB".Send_Cmd_Load_Recipe )
   END_RUNG
   // the same network as SCL:
   "DB_PLC1_MB_Buffer_DB".Send_Cmd_Load_Recipe := "DB_PLC1_Send_To_PLC2_DB".Cmd_Load_Recipe;
END_REGION

REGION Network 10: Modbus TCP Client - Copy Send Heartbeat
   RUNG wire#powerrail
      { S7_GenerateENO := "TRUE" } Move(in := "DB_PLC1_Send_To_PLC2_DB".Heartbeat, out1 => "DB_PLC1_MB_Buffer_DB".Send_Heartbeat)
   END_RUNG
   // the same network as SCL:
   "DB_PLC1_MB_Buffer_DB".Send_Heartbeat := "DB_PLC1_Send_To_PLC2_DB".Heartbeat;
END_REGION

REGION Network 11: PLC1 - Gọi logic khởi tạo recipe mặc định PLC1
   RUNG wire#powerrail
      "FC_Init_Default_Recipe_PLC1"()
   END_RUNG
   // the same network as SCL:
   "FC_Init_Default_Recipe_PLC1"();
END_REGION

REGION Network 12: PLC1 - gọi logic Bồn 1 và Bồn 2
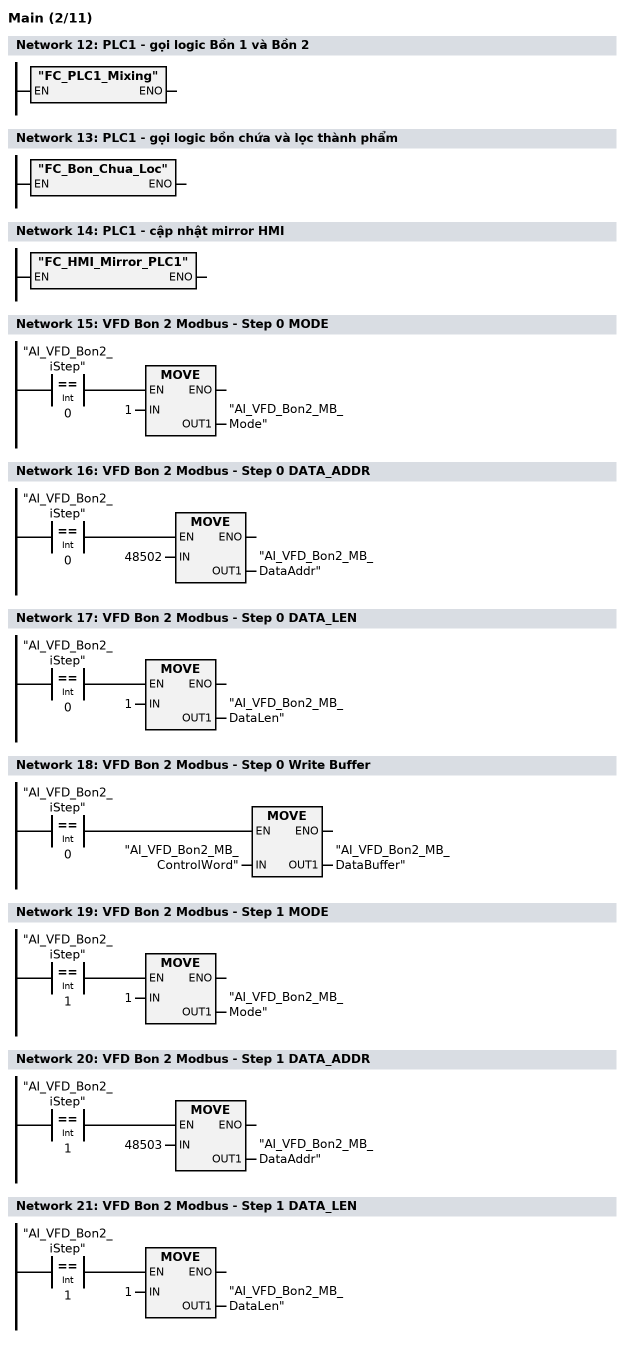
   RUNG wire#powerrail
      "FC_PLC1_Mixing"()
   END_RUNG
   // the same network as SCL:
   "FC_PLC1_Mixing"();
END_REGION

REGION Network 13: PLC1 - gọi logic bồn chứa và lọc thành phẩm
   RUNG wire#powerrail
      "FC_Bon_Chua_Loc"()
   END_RUNG
   // the same network as SCL:
   "FC_Bon_Chua_Loc"();
END_REGION

REGION Network 14: PLC1 - cập nhật mirror HMI
   RUNG wire#powerrail
      "FC_HMI_Mirror_PLC1"()
   END_RUNG
   // the same network as SCL:
   "FC_HMI_Mirror_PLC1"();
END_REGION

REGION Network 15: VFD Bon 2 Modbus - Step 0 MODE
   RUNG wire#powerrail
      { S7_Templates := "SrcType := Int" } EQ_Contact(in1 := "AI_VFD_Bon2_iStep", in2 := 0)
      { S7_GenerateENO := "TRUE" } Move(in := 1, out1 => "AI_VFD_Bon2_MB_Mode")
   END_RUNG
   // the same network as SCL:
   IF "AI_VFD_Bon2_iStep" = 0 THEN "AI_VFD_Bon2_MB_Mode" := 1; END_IF;
END_REGION

REGION Network 16: VFD Bon 2 Modbus - Step 0 DATA_ADDR
   RUNG wire#powerrail
      { S7_Templates := "SrcType := Int" } EQ_Contact(in1 := "AI_VFD_Bon2_iStep", in2 := 0)
      { S7_GenerateENO := "TRUE" } Move(in := 48502, out1 => "AI_VFD_Bon2_MB_DataAddr")
   END_RUNG
   // the same network as SCL:
   IF "AI_VFD_Bon2_iStep" = 0 THEN "AI_VFD_Bon2_MB_DataAddr" := 48502; END_IF;
END_REGION

REGION Network 17: VFD Bon 2 Modbus - Step 0 DATA_LEN
   RUNG wire#powerrail
      { S7_Templates := "SrcType := Int" } EQ_Contact(in1 := "AI_VFD_Bon2_iStep", in2 := 0)
      { S7_GenerateENO := "TRUE" } Move(in := 1, out1 => "AI_VFD_Bon2_MB_DataLen")
   END_RUNG
   // the same network as SCL:
   IF "AI_VFD_Bon2_iStep" = 0 THEN "AI_VFD_Bon2_MB_DataLen" := 1; END_IF;
END_REGION

REGION Network 18: VFD Bon 2 Modbus - Step 0 Write Buffer
   RUNG wire#powerrail
      { S7_Templates := "SrcType := Int" } EQ_Contact(in1 := "AI_VFD_Bon2_iStep", in2 := 0)
      { S7_GenerateENO := "TRUE" } Move(in := "AI_VFD_Bon2_MB_ControlWord", out1 => "AI_VFD_Bon2_MB_DataBuffer")
   END_RUNG
   // the same network as SCL:
   IF "AI_VFD_Bon2_iStep" = 0 THEN "AI_VFD_Bon2_MB_DataBuffer" := "AI_VFD_Bon2_MB_ControlWord"; END_IF;
END_REGION

REGION Network 19: VFD Bon 2 Modbus - Step 1 MODE
   RUNG wire#powerrail
      { S7_Templates := "SrcType := Int" } EQ_Contact(in1 := "AI_VFD_Bon2_iStep", in2 := 1)
      { S7_GenerateENO := "TRUE" } Move(in := 1, out1 => "AI_VFD_Bon2_MB_Mode")
   END_RUNG
   // the same network as SCL:
   IF "AI_VFD_Bon2_iStep" = 1 THEN "AI_VFD_Bon2_MB_Mode" := 1; END_IF;
END_REGION

REGION Network 20: VFD Bon 2 Modbus - Step 1 DATA_ADDR
   RUNG wire#powerrail
      { S7_Templates := "SrcType := Int" } EQ_Contact(in1 := "AI_VFD_Bon2_iStep", in2 := 1)
      { S7_GenerateENO := "TRUE" } Move(in := 48503, out1 => "AI_VFD_Bon2_MB_DataAddr")
   END_RUNG
   // the same network as SCL:
   IF "AI_VFD_Bon2_iStep" = 1 THEN "AI_VFD_Bon2_MB_DataAddr" := 48503; END_IF;
END_REGION

REGION Network 21: VFD Bon 2 Modbus - Step 1 DATA_LEN
   RUNG wire#powerrail
      { S7_Templates := "SrcType := Int" } EQ_Contact(in1 := "AI_VFD_Bon2_iStep", in2 := 1)
      { S7_GenerateENO := "TRUE" } Move(in := 1, out1 => "AI_VFD_Bon2_MB_DataLen")
   END_RUNG
   // the same network as SCL:
   IF "AI_VFD_Bon2_iStep" = 1 THEN "AI_VFD_Bon2_MB_DataLen" := 1; END_IF;
END_REGION

REGION Network 22: VFD Bon 2 Modbus - Step 1 Write Buffer
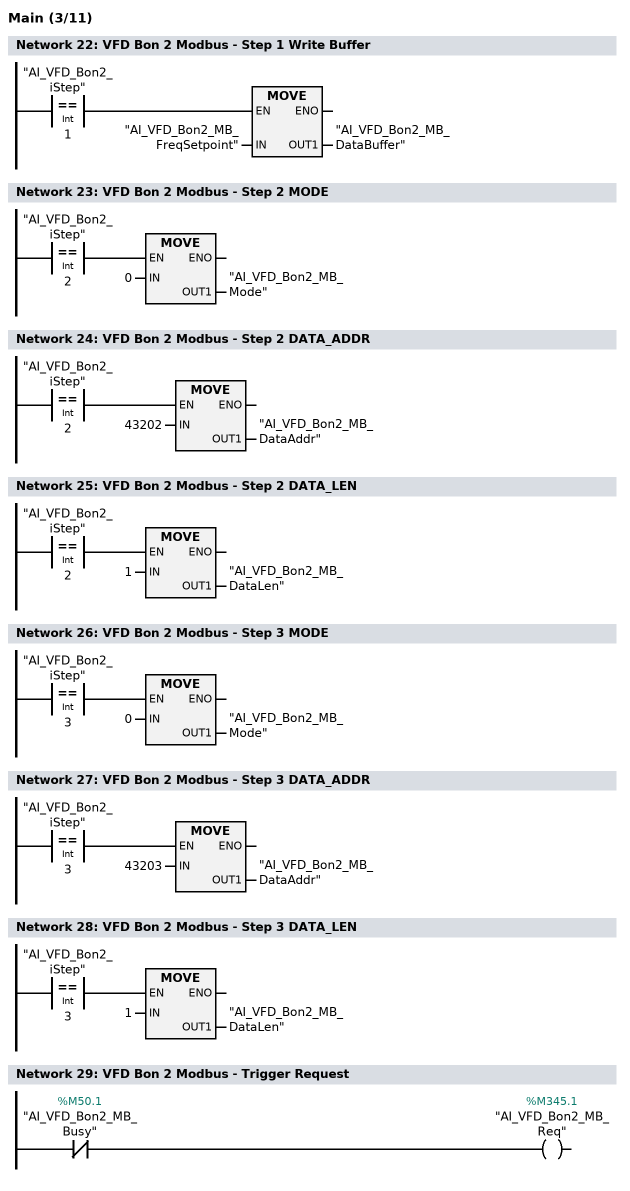
   RUNG wire#powerrail
      { S7_Templates := "SrcType := Int" } EQ_Contact(in1 := "AI_VFD_Bon2_iStep", in2 := 1)
      { S7_GenerateENO := "TRUE" } Move(in := "AI_VFD_Bon2_MB_FreqSetpoint", out1 => "AI_VFD_Bon2_MB_DataBuffer")
   END_RUNG
   // the same network as SCL:
   IF "AI_VFD_Bon2_iStep" = 1 THEN "AI_VFD_Bon2_MB_DataBuffer" := "AI_VFD_Bon2_MB_FreqSetpoint"; END_IF;
END_REGION

REGION Network 23: VFD Bon 2 Modbus - Step 2 MODE
   RUNG wire#powerrail
      { S7_Templates := "SrcType := Int" } EQ_Contact(in1 := "AI_VFD_Bon2_iStep", in2 := 2)
      { S7_GenerateENO := "TRUE" } Move(in := 0, out1 => "AI_VFD_Bon2_MB_Mode")
   END_RUNG
   // the same network as SCL:
   IF "AI_VFD_Bon2_iStep" = 2 THEN "AI_VFD_Bon2_MB_Mode" := 0; END_IF;
END_REGION

REGION Network 24: VFD Bon 2 Modbus - Step 2 DATA_ADDR
   RUNG wire#powerrail
      { S7_Templates := "SrcType := Int" } EQ_Contact(in1 := "AI_VFD_Bon2_iStep", in2 := 2)
      { S7_GenerateENO := "TRUE" } Move(in := 43202, out1 => "AI_VFD_Bon2_MB_DataAddr")
   END_RUNG
   // the same network as SCL:
   IF "AI_VFD_Bon2_iStep" = 2 THEN "AI_VFD_Bon2_MB_DataAddr" := 43202; END_IF;
END_REGION

REGION Network 25: VFD Bon 2 Modbus - Step 2 DATA_LEN
   RUNG wire#powerrail
      { S7_Templates := "SrcType := Int" } EQ_Contact(in1 := "AI_VFD_Bon2_iStep", in2 := 2)
      { S7_GenerateENO := "TRUE" } Move(in := 1, out1 => "AI_VFD_Bon2_MB_DataLen")
   END_RUNG
   // the same network as SCL:
   IF "AI_VFD_Bon2_iStep" = 2 THEN "AI_VFD_Bon2_MB_DataLen" := 1; END_IF;
END_REGION

REGION Network 26: VFD Bon 2 Modbus - Step 3 MODE
   RUNG wire#powerrail
      { S7_Templates := "SrcType := Int" } EQ_Contact(in1 := "AI_VFD_Bon2_iStep", in2 := 3)
      { S7_GenerateENO := "TRUE" } Move(in := 0, out1 => "AI_VFD_Bon2_MB_Mode")
   END_RUNG
   // the same network as SCL:
   IF "AI_VFD_Bon2_iStep" = 3 THEN "AI_VFD_Bon2_MB_Mode" := 0; END_IF;
END_REGION

REGION Network 27: VFD Bon 2 Modbus - Step 3 DATA_ADDR
   RUNG wire#powerrail
      { S7_Templates := "SrcType := Int" } EQ_Contact(in1 := "AI_VFD_Bon2_iStep", in2 := 3)
      { S7_GenerateENO := "TRUE" } Move(in := 43203, out1 => "AI_VFD_Bon2_MB_DataAddr")
   END_RUNG
   // the same network as SCL:
   IF "AI_VFD_Bon2_iStep" = 3 THEN "AI_VFD_Bon2_MB_DataAddr" := 43203; END_IF;
END_REGION

REGION Network 28: VFD Bon 2 Modbus - Step 3 DATA_LEN
   RUNG wire#powerrail
      { S7_Templates := "SrcType := Int" } EQ_Contact(in1 := "AI_VFD_Bon2_iStep", in2 := 3)
      { S7_GenerateENO := "TRUE" } Move(in := 1, out1 => "AI_VFD_Bon2_MB_DataLen")
   END_RUNG
   // the same network as SCL:
   IF "AI_VFD_Bon2_iStep" = 3 THEN "AI_VFD_Bon2_MB_DataLen" := 1; END_IF;
END_REGION

REGION Network 29: VFD Bon 2 Modbus - Trigger Request
   RUNG wire#powerrail
      I_Contact( "AI_VFD_Bon2_MB_Busy" )
      Coil( "AI_VFD_Bon2_MB_Req" )
   END_RUNG
   // the same network as SCL:
   "AI_VFD_Bon2_MB_Req" := NOT "AI_VFD_Bon2_MB_Busy";
END_REGION

REGION Network 30: VFD Bon 2 Modbus - Khoi tao RS-485
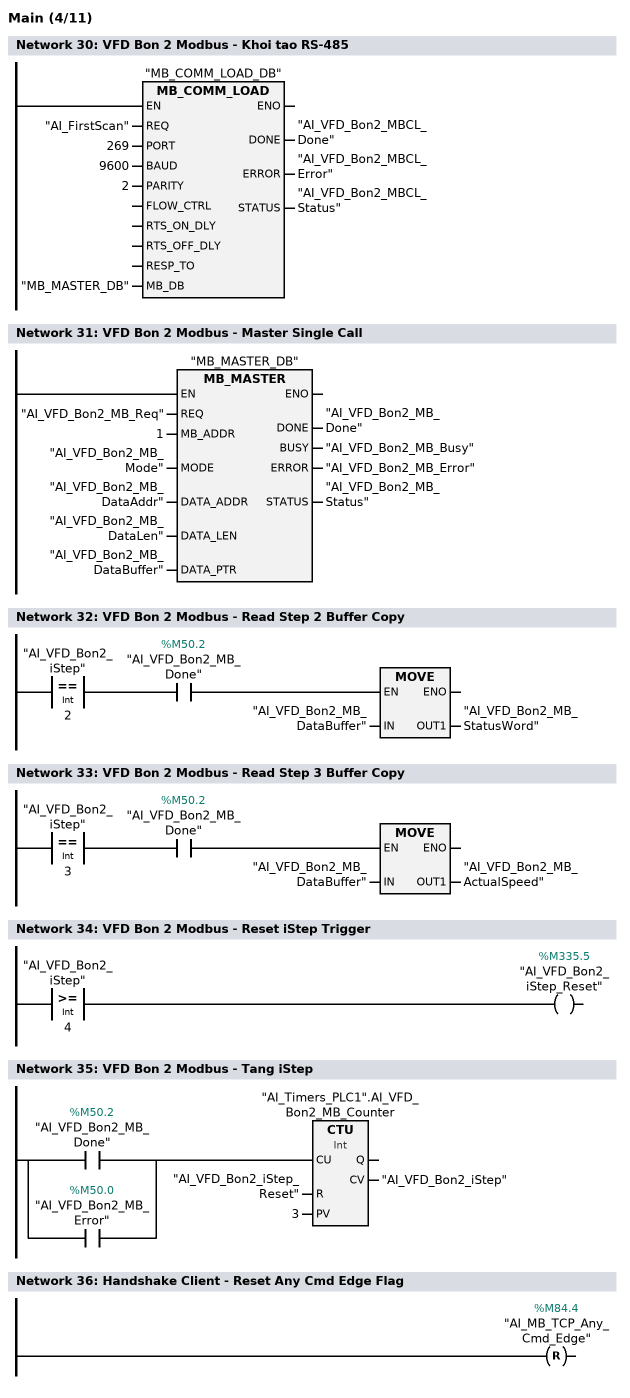
   RUNG wire#powerrail
      "MB_COMM_LOAD_DB".MB_COMM_LOAD(REQ := "AI_FirstScan", PORT := 269, BAUD := 9600, PARITY := 2, FLOW_CTRL :=, RTS_ON_DLY :=, RTS_OFF_DLY :=, RESP_TO :=, MB_DB := "MB_MASTER_DB", DONE => "AI_VFD_Bon2_MBCL_Done", ERROR => "AI_VFD_Bon2_MBCL_Error", STATUS => "AI_VFD_Bon2_MBCL_Status")
   END_RUNG
   // the same network as SCL:
   "MB_COMM_LOAD_DB"(REQ := "AI_FirstScan",   // MB_COMM_LOAD
                     PORT := 269,
                     BAUD := 9600,
                     PARITY := 2,
                     MB_DB := "MB_MASTER_DB",
                     DONE => "AI_VFD_Bon2_MBCL_Done",
                     ERROR => "AI_VFD_Bon2_MBCL_Error",
                     STATUS => "AI_VFD_Bon2_MBCL_Status");
END_REGION

REGION Network 31: VFD Bon 2 Modbus - Master Single Call
   RUNG wire#powerrail
      "MB_MASTER_DB".MB_MASTER(REQ := "AI_VFD_Bon2_MB_Req", MB_ADDR := 1, MODE := "AI_VFD_Bon2_MB_Mode", DATA_ADDR := "AI_VFD_Bon2_MB_DataAddr", DATA_LEN := "AI_VFD_Bon2_MB_DataLen", DATA_PTR := "AI_VFD_Bon2_MB_DataBuffer", DONE => "AI_VFD_Bon2_MB_Done", BUSY => "AI_VFD_Bon2_MB_Busy", ERROR => "AI_VFD_Bon2_MB_Error", STATUS => "AI_VFD_Bon2_MB_Status")
   END_RUNG
   // the same network as SCL:
   "MB_MASTER_DB"(REQ := "AI_VFD_Bon2_MB_Req",   // MB_MASTER
                  MB_ADDR := 1,
                  MODE := "AI_VFD_Bon2_MB_Mode",
                  DATA_ADDR := "AI_VFD_Bon2_MB_DataAddr",
                  DATA_LEN := "AI_VFD_Bon2_MB_DataLen",
                  DATA_PTR := "AI_VFD_Bon2_MB_DataBuffer",
                  DONE => "AI_VFD_Bon2_MB_Done",
                  BUSY => "AI_VFD_Bon2_MB_Busy",
                  ERROR => "AI_VFD_Bon2_MB_Error",
                  STATUS => "AI_VFD_Bon2_MB_Status");
END_REGION

REGION Network 32: VFD Bon 2 Modbus - Read Step 2 Buffer Copy
   RUNG wire#powerrail
      { S7_Templates := "SrcType := Int" } EQ_Contact(in1 := "AI_VFD_Bon2_iStep", in2 := 2)
      Contact( "AI_VFD_Bon2_MB_Done" )
      { S7_GenerateENO := "TRUE" } Move(in := "AI_VFD_Bon2_MB_DataBuffer", out1 => "AI_VFD_Bon2_MB_StatusWord")
   END_RUNG
   // the same network as SCL:
   IF ("AI_VFD_Bon2_iStep" = 2) AND "AI_VFD_Bon2_MB_Done" THEN
       "AI_VFD_Bon2_MB_StatusWord" := "AI_VFD_Bon2_MB_DataBuffer";
   END_IF;
END_REGION

REGION Network 33: VFD Bon 2 Modbus - Read Step 3 Buffer Copy
   RUNG wire#powerrail
      { S7_Templates := "SrcType := Int" } EQ_Contact(in1 := "AI_VFD_Bon2_iStep", in2 := 3)
      Contact( "AI_VFD_Bon2_MB_Done" )
      { S7_GenerateENO := "TRUE" } Move(in := "AI_VFD_Bon2_MB_DataBuffer", out1 => "AI_VFD_Bon2_MB_ActualSpeed")
   END_RUNG
   // the same network as SCL:
   IF ("AI_VFD_Bon2_iStep" = 3) AND "AI_VFD_Bon2_MB_Done" THEN
       "AI_VFD_Bon2_MB_ActualSpeed" := "AI_VFD_Bon2_MB_DataBuffer";
   END_IF;
END_REGION

REGION Network 34: VFD Bon 2 Modbus - Reset iStep Trigger
   RUNG wire#powerrail
      { S7_Templates := "SrcType := Int" } GE_Contact(in1 := "AI_VFD_Bon2_iStep", in2 := 4)
      Coil( "AI_VFD_Bon2_iStep_Reset" )
   END_RUNG
   // the same network as SCL:
   "AI_VFD_Bon2_iStep_Reset" := "AI_VFD_Bon2_iStep" >= 4;
END_REGION

REGION Network 35: VFD Bon 2 Modbus - Tang iStep
   RUNG wire#powerrail
      Contact( "AI_VFD_Bon2_MB_Done" )
      wire#w1
      { S7_Templates := "value_type := Int" } "AI_Timers_PLC1".AI_VFD_Bon2_MB_Counter.CTU(r := "AI_VFD_Bon2_iStep_Reset", pv := 3, cv => "AI_VFD_Bon2_iStep")
   END_RUNG
   RUNG wire#powerrail
      Contact( "AI_VFD_Bon2_MB_Error" )
   END_RUNG wire#w1
   // the same network as SCL:
   "AI_Timers_PLC1".AI_VFD_Bon2_MB_Counter.CTU(CU := "AI_VFD_Bon2_MB_Done" OR "AI_VFD_Bon2_MB_Error",
                           R := "AI_VFD_Bon2_iStep_Reset",
                           PV := 3,
                           CV => "AI_VFD_Bon2_iStep");
END_REGION

REGION Network 36: Handshake Client - Reset Any Cmd Edge Flag
   RUNG wire#powerrail
      R_Coil( "AI_MB_TCP_Any_Cmd_Edge" )
   END_RUNG
   // the same network as SCL:
   "AI_MB_TCP_Any_Cmd_Edge" := FALSE;
END_REGION

REGION Network 37: Handshake Client - Start Edge
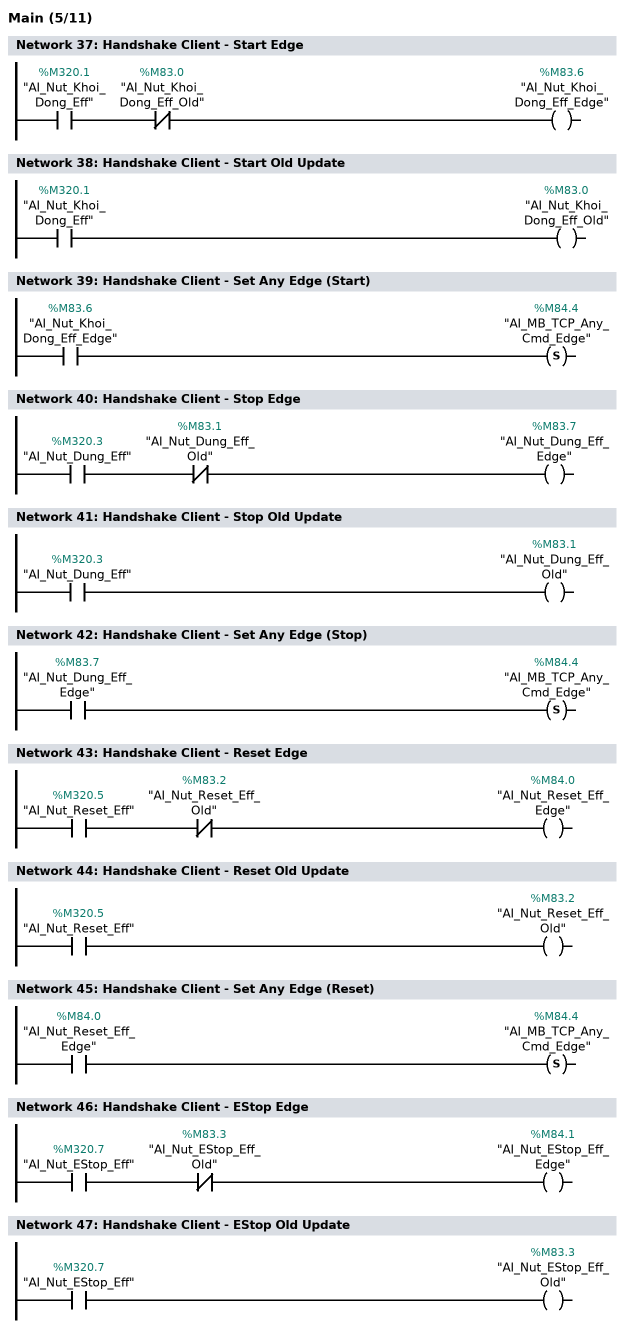
   RUNG wire#powerrail
      Contact( "AI_Nut_Khoi_Dong_Eff" )
      I_Contact( "AI_Nut_Khoi_Dong_Eff_Old" )
      Coil( "AI_Nut_Khoi_Dong_Eff_Edge" )
   END_RUNG
   // the same network as SCL:
   "AI_Nut_Khoi_Dong_Eff_Edge" := "AI_Nut_Khoi_Dong_Eff" AND NOT "AI_Nut_Khoi_Dong_Eff_Old";
END_REGION

REGION Network 38: Handshake Client - Start Old Update
   RUNG wire#powerrail
      Contact( "AI_Nut_Khoi_Dong_Eff" )
      Coil( "AI_Nut_Khoi_Dong_Eff_Old" )
   END_RUNG
   // the same network as SCL:
   "AI_Nut_Khoi_Dong_Eff_Old" := "AI_Nut_Khoi_Dong_Eff";
END_REGION

REGION Network 39: Handshake Client - Set Any Edge (Start)
   RUNG wire#powerrail
      Contact( "AI_Nut_Khoi_Dong_Eff_Edge" )
      S_Coil( "AI_MB_TCP_Any_Cmd_Edge" )
   END_RUNG
   // the same network as SCL:
   IF "AI_Nut_Khoi_Dong_Eff_Edge" THEN "AI_MB_TCP_Any_Cmd_Edge" := TRUE; END_IF;
END_REGION

REGION Network 40: Handshake Client - Stop Edge
   RUNG wire#powerrail
      Contact( "AI_Nut_Dung_Eff" )
      I_Contact( "AI_Nut_Dung_Eff_Old" )
      Coil( "AI_Nut_Dung_Eff_Edge" )
   END_RUNG
   // the same network as SCL:
   "AI_Nut_Dung_Eff_Edge" := "AI_Nut_Dung_Eff" AND NOT "AI_Nut_Dung_Eff_Old";
END_REGION

REGION Network 41: Handshake Client - Stop Old Update
   RUNG wire#powerrail
      Contact( "AI_Nut_Dung_Eff" )
      Coil( "AI_Nut_Dung_Eff_Old" )
   END_RUNG
   // the same network as SCL:
   "AI_Nut_Dung_Eff_Old" := "AI_Nut_Dung_Eff";
END_REGION

REGION Network 42: Handshake Client - Set Any Edge (Stop)
   RUNG wire#powerrail
      Contact( "AI_Nut_Dung_Eff_Edge" )
      S_Coil( "AI_MB_TCP_Any_Cmd_Edge" )
   END_RUNG
   // the same network as SCL:
   IF "AI_Nut_Dung_Eff_Edge" THEN "AI_MB_TCP_Any_Cmd_Edge" := TRUE; END_IF;
END_REGION

REGION Network 43: Handshake Client - Reset Edge
   RUNG wire#powerrail
      Contact( "AI_Nut_Reset_Eff" )
      I_Contact( "AI_Nut_Reset_Eff_Old" )
      Coil( "AI_Nut_Reset_Eff_Edge" )
   END_RUNG
   // the same network as SCL:
   "AI_Nut_Reset_Eff_Edge" := "AI_Nut_Reset_Eff" AND NOT "AI_Nut_Reset_Eff_Old";
END_REGION

REGION Network 44: Handshake Client - Reset Old Update
   RUNG wire#powerrail
      Contact( "AI_Nut_Reset_Eff" )
      Coil( "AI_Nut_Reset_Eff_Old" )
   END_RUNG
   // the same network as SCL:
   "AI_Nut_Reset_Eff_Old" := "AI_Nut_Reset_Eff";
END_REGION

REGION Network 45: Handshake Client - Set Any Edge (Reset)
   RUNG wire#powerrail
      Contact( "AI_Nut_Reset_Eff_Edge" )
      S_Coil( "AI_MB_TCP_Any_Cmd_Edge" )
   END_RUNG
   // the same network as SCL:
   IF "AI_Nut_Reset_Eff_Edge" THEN "AI_MB_TCP_Any_Cmd_Edge" := TRUE; END_IF;
END_REGION

REGION Network 46: Handshake Client - EStop Edge
   RUNG wire#powerrail
      Contact( "AI_Nut_EStop_Eff" )
      I_Contact( "AI_Nut_EStop_Eff_Old" )
      Coil( "AI_Nut_EStop_Eff_Edge" )
   END_RUNG
   // the same network as SCL:
   "AI_Nut_EStop_Eff_Edge" := "AI_Nut_EStop_Eff" AND NOT "AI_Nut_EStop_Eff_Old";
END_REGION

REGION Network 47: Handshake Client - EStop Old Update
   RUNG wire#powerrail
      Contact( "AI_Nut_EStop_Eff" )
      Coil( "AI_Nut_EStop_Eff_Old" )
   END_RUNG
   // the same network as SCL:
   "AI_Nut_EStop_Eff_Old" := "AI_Nut_EStop_Eff";
END_REGION

REGION Network 48: Handshake Client - Set Any Edge (EStop)
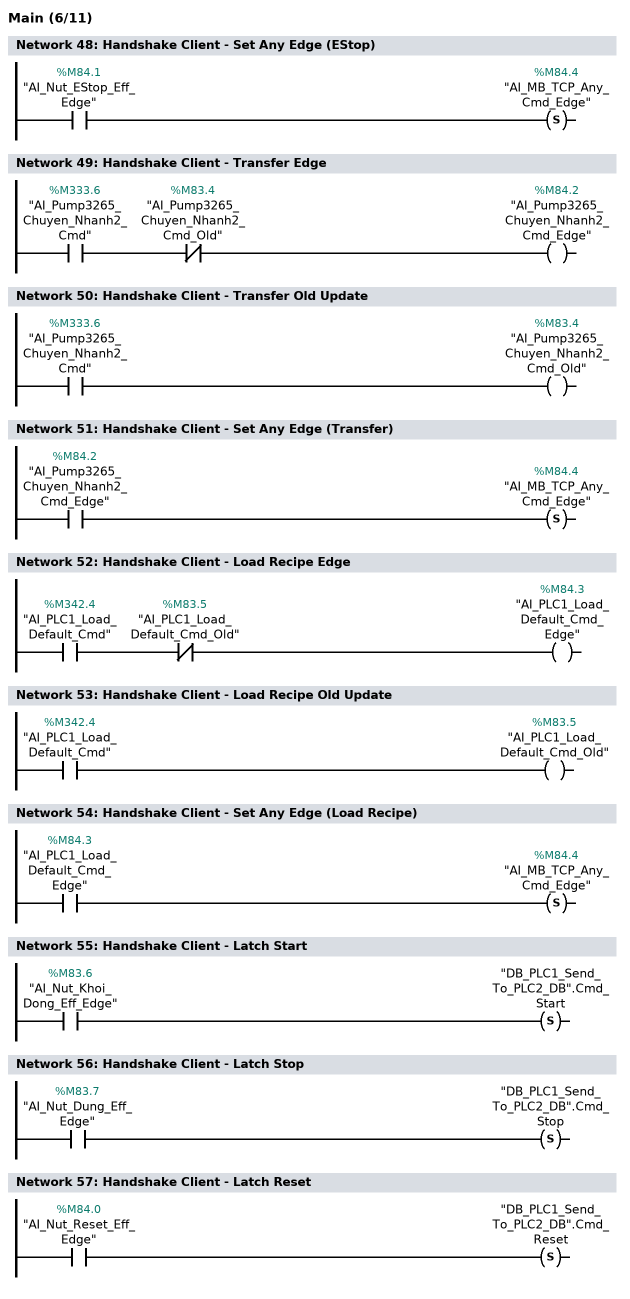
   RUNG wire#powerrail
      Contact( "AI_Nut_EStop_Eff_Edge" )
      S_Coil( "AI_MB_TCP_Any_Cmd_Edge" )
   END_RUNG
   // the same network as SCL:
   IF "AI_Nut_EStop_Eff_Edge" THEN "AI_MB_TCP_Any_Cmd_Edge" := TRUE; END_IF;
END_REGION

REGION Network 49: Handshake Client - Transfer Edge
   RUNG wire#powerrail
      Contact( "AI_Pump3265_Chuyen_Nhanh2_Cmd" )
      I_Contact( "AI_Pump3265_Chuyen_Nhanh2_Cmd_Old" )
      Coil( "AI_Pump3265_Chuyen_Nhanh2_Cmd_Edge" )
   END_RUNG
   // the same network as SCL:
   "AI_Pump3265_Chuyen_Nhanh2_Cmd_Edge" := "AI_Pump3265_Chuyen_Nhanh2_Cmd" AND NOT "AI_Pump3265_Chuyen_Nhanh2_Cmd_Old";
END_REGION

REGION Network 50: Handshake Client - Transfer Old Update
   RUNG wire#powerrail
      Contact( "AI_Pump3265_Chuyen_Nhanh2_Cmd" )
      Coil( "AI_Pump3265_Chuyen_Nhanh2_Cmd_Old" )
   END_RUNG
   // the same network as SCL:
   "AI_Pump3265_Chuyen_Nhanh2_Cmd_Old" := "AI_Pump3265_Chuyen_Nhanh2_Cmd";
END_REGION

REGION Network 51: Handshake Client - Set Any Edge (Transfer)
   RUNG wire#powerrail
      Contact( "AI_Pump3265_Chuyen_Nhanh2_Cmd_Edge" )
      S_Coil( "AI_MB_TCP_Any_Cmd_Edge" )
   END_RUNG
   // the same network as SCL:
   IF "AI_Pump3265_Chuyen_Nhanh2_Cmd_Edge" THEN "AI_MB_TCP_Any_Cmd_Edge" := TRUE; END_IF;
END_REGION

REGION Network 52: Handshake Client - Load Recipe Edge
   RUNG wire#powerrail
      Contact( "AI_PLC1_Load_Default_Cmd" )
      I_Contact( "AI_PLC1_Load_Default_Cmd_Old" )
      Coil( "AI_PLC1_Load_Default_Cmd_Edge" )
   END_RUNG
   // the same network as SCL:
   "AI_PLC1_Load_Default_Cmd_Edge" := "AI_PLC1_Load_Default_Cmd" AND NOT "AI_PLC1_Load_Default_Cmd_Old";
END_REGION

REGION Network 53: Handshake Client - Load Recipe Old Update
   RUNG wire#powerrail
      Contact( "AI_PLC1_Load_Default_Cmd" )
      Coil( "AI_PLC1_Load_Default_Cmd_Old" )
   END_RUNG
   // the same network as SCL:
   "AI_PLC1_Load_Default_Cmd_Old" := "AI_PLC1_Load_Default_Cmd";
END_REGION

REGION Network 54: Handshake Client - Set Any Edge (Load Recipe)
   RUNG wire#powerrail
      Contact( "AI_PLC1_Load_Default_Cmd_Edge" )
      S_Coil( "AI_MB_TCP_Any_Cmd_Edge" )
   END_RUNG
   // the same network as SCL:
   IF "AI_PLC1_Load_Default_Cmd_Edge" THEN "AI_MB_TCP_Any_Cmd_Edge" := TRUE; END_IF;
END_REGION

REGION Network 55: Handshake Client - Latch Start
   RUNG wire#powerrail
      Contact( "AI_Nut_Khoi_Dong_Eff_Edge" )
      S_Coil( "DB_PLC1_Send_To_PLC2_DB".Cmd_Start )
   END_RUNG
   // the same network as SCL:
   IF "AI_Nut_Khoi_Dong_Eff_Edge" THEN "DB_PLC1_Send_To_PLC2_DB".Cmd_Start := TRUE; END_IF;
END_REGION

REGION Network 56: Handshake Client - Latch Stop
   RUNG wire#powerrail
      Contact( "AI_Nut_Dung_Eff_Edge" )
      S_Coil( "DB_PLC1_Send_To_PLC2_DB".Cmd_Stop )
   END_RUNG
   // the same network as SCL:
   IF "AI_Nut_Dung_Eff_Edge" THEN "DB_PLC1_Send_To_PLC2_DB".Cmd_Stop := TRUE; END_IF;
END_REGION

REGION Network 57: Handshake Client - Latch Reset
   RUNG wire#powerrail
      Contact( "AI_Nut_Reset_Eff_Edge" )
      S_Coil( "DB_PLC1_Send_To_PLC2_DB".Cmd_Reset )
   END_RUNG
   // the same network as SCL:
   IF "AI_Nut_Reset_Eff_Edge" THEN "DB_PLC1_Send_To_PLC2_DB".Cmd_Reset := TRUE; END_IF;
END_REGION

REGION Network 58: Handshake Client - Latch EStop
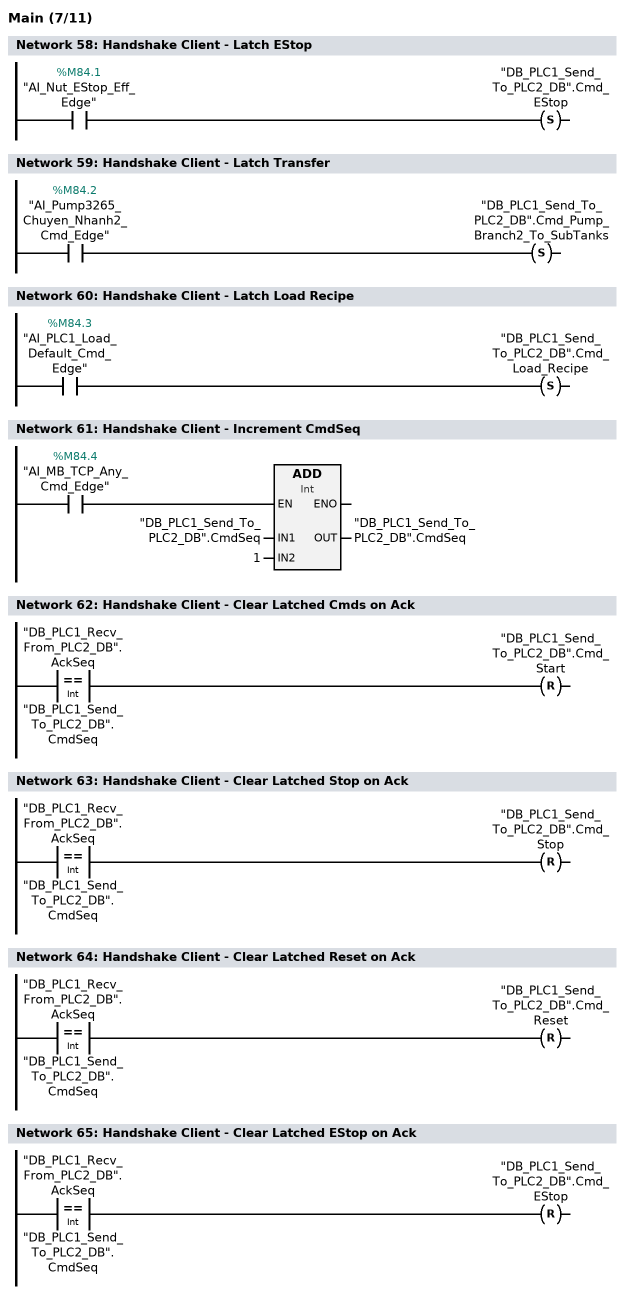
   RUNG wire#powerrail
      Contact( "AI_Nut_EStop_Eff_Edge" )
      S_Coil( "DB_PLC1_Send_To_PLC2_DB".Cmd_EStop )
   END_RUNG
   // the same network as SCL:
   IF "AI_Nut_EStop_Eff_Edge" THEN "DB_PLC1_Send_To_PLC2_DB".Cmd_EStop := TRUE; END_IF;
END_REGION

REGION Network 59: Handshake Client - Latch Transfer
   RUNG wire#powerrail
      Contact( "AI_Pump3265_Chuyen_Nhanh2_Cmd_Edge" )
      S_Coil( "DB_PLC1_Send_To_PLC2_DB".Cmd_Pump_Branch2_To_SubTanks )
   END_RUNG
   // the same network as SCL:
   IF "AI_Pump3265_Chuyen_Nhanh2_Cmd_Edge" THEN
       "DB_PLC1_Send_To_PLC2_DB".Cmd_Pump_Branch2_To_SubTanks := TRUE;
   END_IF;
END_REGION

REGION Network 60: Handshake Client - Latch Load Recipe
   RUNG wire#powerrail
      Contact( "AI_PLC1_Load_Default_Cmd_Edge" )
      S_Coil( "DB_PLC1_Send_To_PLC2_DB".Cmd_Load_Recipe )
   END_RUNG
   // the same network as SCL:
   IF "AI_PLC1_Load_Default_Cmd_Edge" THEN "DB_PLC1_Send_To_PLC2_DB".Cmd_Load_Recipe := TRUE; END_IF;
END_REGION

REGION Network 61: Handshake Client - Increment CmdSeq
   RUNG wire#powerrail
      Contact( "AI_MB_TCP_Any_Cmd_Edge" )
      { S7_Templates := "SrcType := Int"; S7_GenerateENO := "TRUE" } Add(in1 := "DB_PLC1_Send_To_PLC2_DB".CmdSeq, in2 := 1, out => "DB_PLC1_Send_To_PLC2_DB".CmdSeq)
   END_RUNG
   // the same network as SCL:
   IF "AI_MB_TCP_Any_Cmd_Edge" THEN
       "DB_PLC1_Send_To_PLC2_DB".CmdSeq := "DB_PLC1_Send_To_PLC2_DB".CmdSeq + 1;
   END_IF;
END_REGION

REGION Network 62: Handshake Client - Clear Latched Cmds on Ack
   RUNG wire#powerrail
      { S7_Templates := "SrcType := Int" } EQ_Contact(in1 := "DB_PLC1_Recv_From_PLC2_DB".AckSeq, in2 := "DB_PLC1_Send_To_PLC2_DB".CmdSeq)
      R_Coil( "DB_PLC1_Send_To_PLC2_DB".Cmd_Start )
   END_RUNG
   // the same network as SCL:
   IF "DB_PLC1_Recv_From_PLC2_DB".AckSeq = "DB_PLC1_Send_To_PLC2_DB".CmdSeq THEN
       "DB_PLC1_Send_To_PLC2_DB".Cmd_Start := FALSE;
   END_IF;
END_REGION

REGION Network 63: Handshake Client - Clear Latched Stop on Ack
   RUNG wire#powerrail
      { S7_Templates := "SrcType := Int" } EQ_Contact(in1 := "DB_PLC1_Recv_From_PLC2_DB".AckSeq, in2 := "DB_PLC1_Send_To_PLC2_DB".CmdSeq)
      R_Coil( "DB_PLC1_Send_To_PLC2_DB".Cmd_Stop )
   END_RUNG
   // the same network as SCL:
   IF "DB_PLC1_Recv_From_PLC2_DB".AckSeq = "DB_PLC1_Send_To_PLC2_DB".CmdSeq THEN
       "DB_PLC1_Send_To_PLC2_DB".Cmd_Stop := FALSE;
   END_IF;
END_REGION

REGION Network 64: Handshake Client - Clear Latched Reset on Ack
   RUNG wire#powerrail
      { S7_Templates := "SrcType := Int" } EQ_Contact(in1 := "DB_PLC1_Recv_From_PLC2_DB".AckSeq, in2 := "DB_PLC1_Send_To_PLC2_DB".CmdSeq)
      R_Coil( "DB_PLC1_Send_To_PLC2_DB".Cmd_Reset )
   END_RUNG
   // the same network as SCL:
   IF "DB_PLC1_Recv_From_PLC2_DB".AckSeq = "DB_PLC1_Send_To_PLC2_DB".CmdSeq THEN
       "DB_PLC1_Send_To_PLC2_DB".Cmd_Reset := FALSE;
   END_IF;
END_REGION

REGION Network 65: Handshake Client - Clear Latched EStop on Ack
   RUNG wire#powerrail
      { S7_Templates := "SrcType := Int" } EQ_Contact(in1 := "DB_PLC1_Recv_From_PLC2_DB".AckSeq, in2 := "DB_PLC1_Send_To_PLC2_DB".CmdSeq)
      R_Coil( "DB_PLC1_Send_To_PLC2_DB".Cmd_EStop )
   END_RUNG
   // the same network as SCL:
   IF "DB_PLC1_Recv_From_PLC2_DB".AckSeq = "DB_PLC1_Send_To_PLC2_DB".CmdSeq THEN
       "DB_PLC1_Send_To_PLC2_DB".Cmd_EStop := FALSE;
   END_IF;
END_REGION

REGION Network 66: Handshake Client - Clear Latched Transfer on Ack
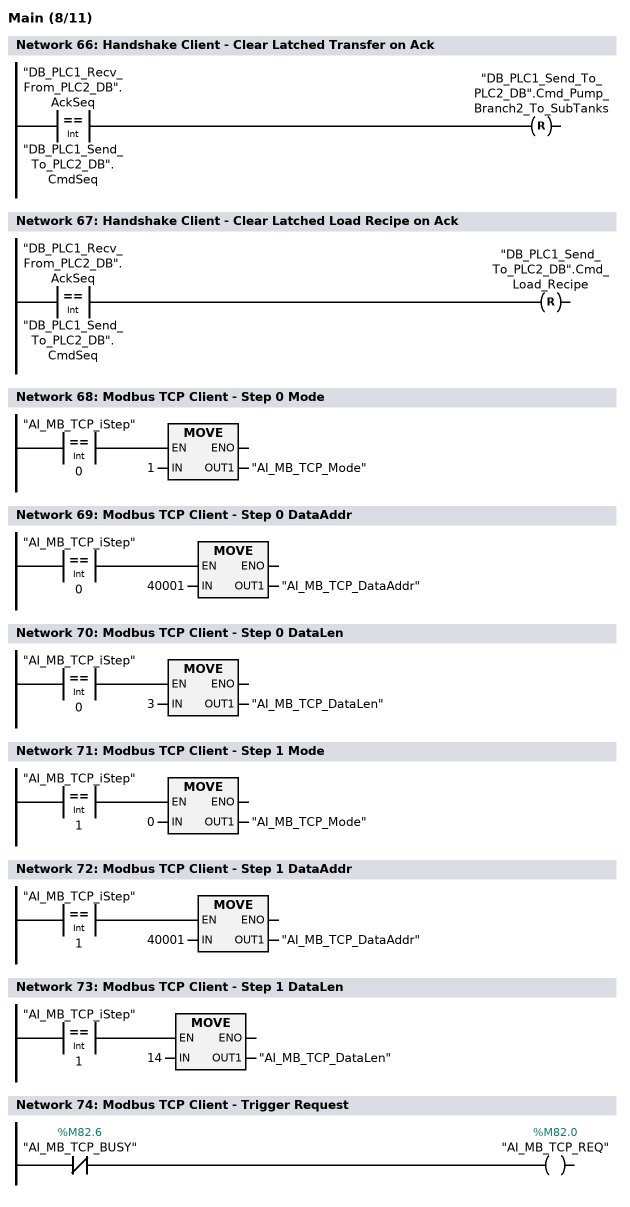
   RUNG wire#powerrail
      { S7_Templates := "SrcType := Int" } EQ_Contact(in1 := "DB_PLC1_Recv_From_PLC2_DB".AckSeq, in2 := "DB_PLC1_Send_To_PLC2_DB".CmdSeq)
      R_Coil( "DB_PLC1_Send_To_PLC2_DB".Cmd_Pump_Branch2_To_SubTanks )
   END_RUNG
   // the same network as SCL:
   IF "DB_PLC1_Recv_From_PLC2_DB".AckSeq = "DB_PLC1_Send_To_PLC2_DB".CmdSeq THEN
       "DB_PLC1_Send_To_PLC2_DB".Cmd_Pump_Branch2_To_SubTanks := FALSE;
   END_IF;
END_REGION

REGION Network 67: Handshake Client - Clear Latched Load Recipe on Ack
   RUNG wire#powerrail
      { S7_Templates := "SrcType := Int" } EQ_Contact(in1 := "DB_PLC1_Recv_From_PLC2_DB".AckSeq, in2 := "DB_PLC1_Send_To_PLC2_DB".CmdSeq)
      R_Coil( "DB_PLC1_Send_To_PLC2_DB".Cmd_Load_Recipe )
   END_RUNG
   // the same network as SCL:
   IF "DB_PLC1_Recv_From_PLC2_DB".AckSeq = "DB_PLC1_Send_To_PLC2_DB".CmdSeq THEN
       "DB_PLC1_Send_To_PLC2_DB".Cmd_Load_Recipe := FALSE;
   END_IF;
END_REGION

REGION Network 68: Modbus TCP Client - Step 0 Mode
   RUNG wire#powerrail
      { S7_Templates := "SrcType := Int" } EQ_Contact(in1 := "AI_MB_TCP_iStep", in2 := 0)
      { S7_GenerateENO := "TRUE" } Move(in := 1, out1 => "AI_MB_TCP_Mode")
   END_RUNG
   // the same network as SCL:
   IF "AI_MB_TCP_iStep" = 0 THEN "AI_MB_TCP_Mode" := 1; END_IF;
END_REGION

REGION Network 69: Modbus TCP Client - Step 0 DataAddr
   RUNG wire#powerrail
      { S7_Templates := "SrcType := Int" } EQ_Contact(in1 := "AI_MB_TCP_iStep", in2 := 0)
      { S7_GenerateENO := "TRUE" } Move(in := 40001, out1 => "AI_MB_TCP_DataAddr")
   END_RUNG
   // the same network as SCL:
   IF "AI_MB_TCP_iStep" = 0 THEN "AI_MB_TCP_DataAddr" := 40001; END_IF;
END_REGION

REGION Network 70: Modbus TCP Client - Step 0 DataLen
   RUNG wire#powerrail
      { S7_Templates := "SrcType := Int" } EQ_Contact(in1 := "AI_MB_TCP_iStep", in2 := 0)
      { S7_GenerateENO := "TRUE" } Move(in := 3, out1 => "AI_MB_TCP_DataLen")
   END_RUNG
   // the same network as SCL:
   IF "AI_MB_TCP_iStep" = 0 THEN "AI_MB_TCP_DataLen" := 3; END_IF;
END_REGION

REGION Network 71: Modbus TCP Client - Step 1 Mode
   RUNG wire#powerrail
      { S7_Templates := "SrcType := Int" } EQ_Contact(in1 := "AI_MB_TCP_iStep", in2 := 1)
      { S7_GenerateENO := "TRUE" } Move(in := 0, out1 => "AI_MB_TCP_Mode")
   END_RUNG
   // the same network as SCL:
   IF "AI_MB_TCP_iStep" = 1 THEN "AI_MB_TCP_Mode" := 0; END_IF;
END_REGION

REGION Network 72: Modbus TCP Client - Step 1 DataAddr
   RUNG wire#powerrail
      { S7_Templates := "SrcType := Int" } EQ_Contact(in1 := "AI_MB_TCP_iStep", in2 := 1)
      { S7_GenerateENO := "TRUE" } Move(in := 40001, out1 => "AI_MB_TCP_DataAddr")
   END_RUNG
   // the same network as SCL:
   IF "AI_MB_TCP_iStep" = 1 THEN "AI_MB_TCP_DataAddr" := 40001; END_IF;
END_REGION

REGION Network 73: Modbus TCP Client - Step 1 DataLen
   RUNG wire#powerrail
      { S7_Templates := "SrcType := Int" } EQ_Contact(in1 := "AI_MB_TCP_iStep", in2 := 1)
      { S7_GenerateENO := "TRUE" } Move(in := 14, out1 => "AI_MB_TCP_DataLen")
   END_RUNG
   // the same network as SCL:
   IF "AI_MB_TCP_iStep" = 1 THEN "AI_MB_TCP_DataLen" := 14; END_IF;
END_REGION

REGION Network 74: Modbus TCP Client - Trigger Request
   RUNG wire#powerrail
      I_Contact( "AI_MB_TCP_BUSY" )
      Coil( "AI_MB_TCP_REQ" )
   END_RUNG
   // the same network as SCL:
   "AI_MB_TCP_REQ" := NOT "AI_MB_TCP_BUSY";
END_REGION

REGION Network 75: Modbus TCP Client - Call MB_CLIENT
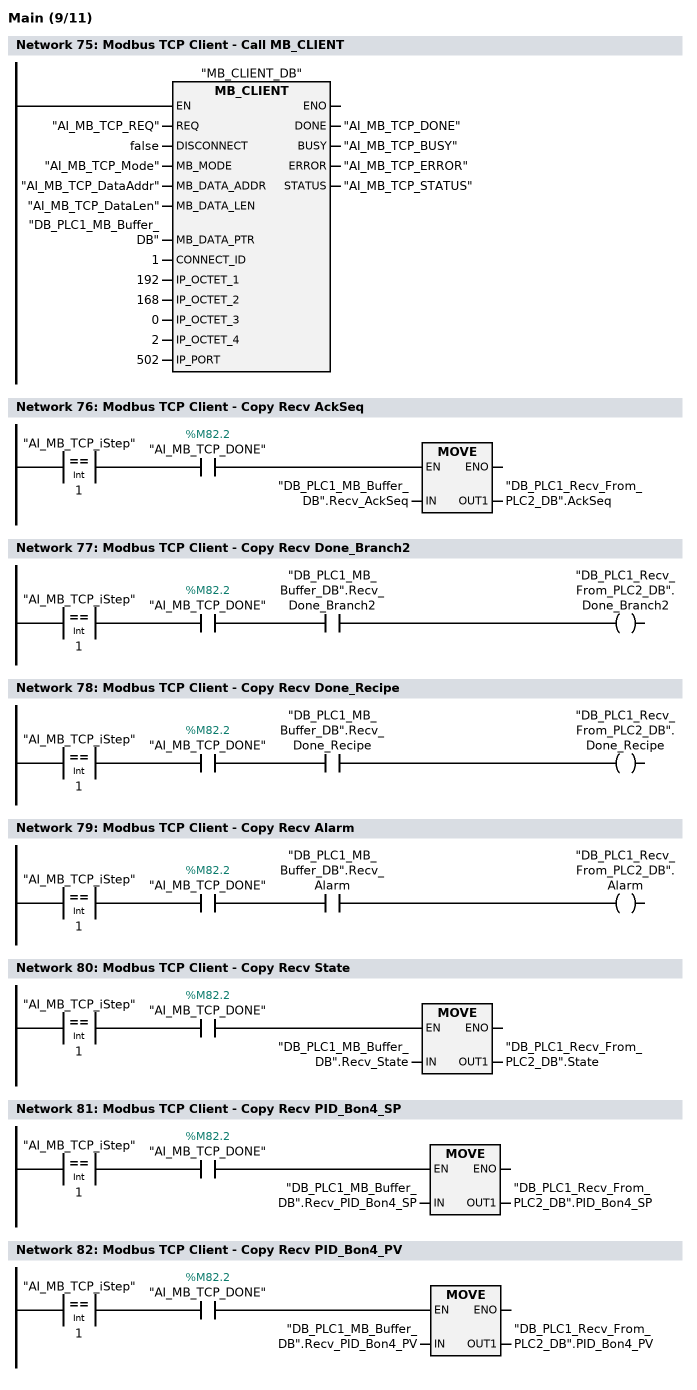
   RUNG wire#powerrail
      { S7_Templates := "[card1200 := 1, card1500 := 0]" } "MB_CLIENT_DB".MB_CLIENT(REQ := "AI_MB_TCP_REQ", DISCONNECT := false, MB_MODE := "AI_MB_TCP_Mode", MB_DATA_ADDR := "AI_MB_TCP_DataAddr", MB_DATA_LEN := "AI_MB_TCP_DataLen", MB_DATA_PTR := "DB_PLC1_MB_Buffer_DB", CONNECT_ID := 1, IP_OCTET_1 := 192, IP_OCTET_2 := 168, IP_OCTET_3 := 0, IP_OCTET_4 := 2, IP_PORT := 502, DONE => "AI_MB_TCP_DONE", BUSY => "AI_MB_TCP_BUSY", ERROR => "AI_MB_TCP_ERROR", STATUS => "AI_MB_TCP_STATUS")
   END_RUNG
   // the same network as SCL:
   "MB_CLIENT_DB"(REQ := "AI_MB_TCP_REQ",   // MB_CLIENT
                  DISCONNECT := false,
                  MB_MODE := "AI_MB_TCP_Mode",
                  MB_DATA_ADDR := "AI_MB_TCP_DataAddr",
                  MB_DATA_LEN := "AI_MB_TCP_DataLen",
                  MB_DATA_PTR := "DB_PLC1_MB_Buffer_DB",
                  CONNECT_ID := 1,
                  IP_OCTET_1 := 192,
                  IP_OCTET_2 := 168,
                  IP_OCTET_3 := 0,
                  IP_OCTET_4 := 2,
                  IP_PORT := 502,
                  DONE => "AI_MB_TCP_DONE",
                  BUSY => "AI_MB_TCP_BUSY",
                  ERROR => "AI_MB_TCP_ERROR",
                  STATUS => "AI_MB_TCP_STATUS");
END_REGION

REGION Network 76: Modbus TCP Client - Copy Recv AckSeq
   RUNG wire#powerrail
      { S7_Templates := "SrcType := Int" } EQ_Contact(in1 := "AI_MB_TCP_iStep", in2 := 1)
      Contact( "AI_MB_TCP_DONE" )
      { S7_GenerateENO := "TRUE" } Move(in := "DB_PLC1_MB_Buffer_DB".Recv_AckSeq, out1 => "DB_PLC1_Recv_From_PLC2_DB".AckSeq)
   END_RUNG
   // the same network as SCL:
   IF ("AI_MB_TCP_iStep" = 1) AND "AI_MB_TCP_DONE" THEN
       "DB_PLC1_Recv_From_PLC2_DB".AckSeq := "DB_PLC1_MB_Buffer_DB".Recv_AckSeq;
   END_IF;
END_REGION

REGION Network 77: Modbus TCP Client - Copy Recv Done_Branch2
   RUNG wire#powerrail
      { S7_Templates := "SrcType := Int" } EQ_Contact(in1 := "AI_MB_TCP_iStep", in2 := 1)
      Contact( "AI_MB_TCP_DONE" )
      Contact( "DB_PLC1_MB_Buffer_DB".Recv_Done_Branch2 )
      Coil( "DB_PLC1_Recv_From_PLC2_DB".Done_Branch2 )
   END_RUNG
   // the same network as SCL:
   "DB_PLC1_Recv_From_PLC2_DB".Done_Branch2 := ("AI_MB_TCP_iStep" = 1) AND "AI_MB_TCP_DONE" AND "DB_PLC1_MB_Buffer_DB".Recv_Done_Branch2;
END_REGION

REGION Network 78: Modbus TCP Client - Copy Recv Done_Recipe
   RUNG wire#powerrail
      { S7_Templates := "SrcType := Int" } EQ_Contact(in1 := "AI_MB_TCP_iStep", in2 := 1)
      Contact( "AI_MB_TCP_DONE" )
      Contact( "DB_PLC1_MB_Buffer_DB".Recv_Done_Recipe )
      Coil( "DB_PLC1_Recv_From_PLC2_DB".Done_Recipe )
   END_RUNG
   // the same network as SCL:
   "DB_PLC1_Recv_From_PLC2_DB".Done_Recipe := ("AI_MB_TCP_iStep" = 1) AND "AI_MB_TCP_DONE" AND "DB_PLC1_MB_Buffer_DB".Recv_Done_Recipe;
END_REGION

REGION Network 79: Modbus TCP Client - Copy Recv Alarm
   RUNG wire#powerrail
      { S7_Templates := "SrcType := Int" } EQ_Contact(in1 := "AI_MB_TCP_iStep", in2 := 1)
      Contact( "AI_MB_TCP_DONE" )
      Contact( "DB_PLC1_MB_Buffer_DB".Recv_Alarm )
      Coil( "DB_PLC1_Recv_From_PLC2_DB".Alarm )
   END_RUNG
   // the same network as SCL:
   "DB_PLC1_Recv_From_PLC2_DB".Alarm := ("AI_MB_TCP_iStep" = 1) AND "AI_MB_TCP_DONE" AND "DB_PLC1_MB_Buffer_DB".Recv_Alarm;
END_REGION

REGION Network 80: Modbus TCP Client - Copy Recv State
   RUNG wire#powerrail
      { S7_Templates := "SrcType := Int" } EQ_Contact(in1 := "AI_MB_TCP_iStep", in2 := 1)
      Contact( "AI_MB_TCP_DONE" )
      { S7_GenerateENO := "TRUE" } Move(in := "DB_PLC1_MB_Buffer_DB".Recv_State, out1 => "DB_PLC1_Recv_From_PLC2_DB".State)
   END_RUNG
   // the same network as SCL:
   IF ("AI_MB_TCP_iStep" = 1) AND "AI_MB_TCP_DONE" THEN
       "DB_PLC1_Recv_From_PLC2_DB".State := "DB_PLC1_MB_Buffer_DB".Recv_State;
   END_IF;
END_REGION

REGION Network 81: Modbus TCP Client - Copy Recv PID_Bon4_SP
   RUNG wire#powerrail
      { S7_Templates := "SrcType := Int" } EQ_Contact(in1 := "AI_MB_TCP_iStep", in2 := 1)
      Contact( "AI_MB_TCP_DONE" )
      { S7_GenerateENO := "TRUE" } Move(in := "DB_PLC1_MB_Buffer_DB".Recv_PID_Bon4_SP, out1 => "DB_PLC1_Recv_From_PLC2_DB".PID_Bon4_SP)
   END_RUNG
   // the same network as SCL:
   IF ("AI_MB_TCP_iStep" = 1) AND "AI_MB_TCP_DONE" THEN
       "DB_PLC1_Recv_From_PLC2_DB".PID_Bon4_SP := "DB_PLC1_MB_Buffer_DB".Recv_PID_Bon4_SP;
   END_IF;
END_REGION

REGION Network 82: Modbus TCP Client - Copy Recv PID_Bon4_PV
   RUNG wire#powerrail
      { S7_Templates := "SrcType := Int" } EQ_Contact(in1 := "AI_MB_TCP_iStep", in2 := 1)
      Contact( "AI_MB_TCP_DONE" )
      { S7_GenerateENO := "TRUE" } Move(in := "DB_PLC1_MB_Buffer_DB".Recv_PID_Bon4_PV, out1 => "DB_PLC1_Recv_From_PLC2_DB".PID_Bon4_PV)
   END_RUNG
   // the same network as SCL:
   IF ("AI_MB_TCP_iStep" = 1) AND "AI_MB_TCP_DONE" THEN
       "DB_PLC1_Recv_From_PLC2_DB".PID_Bon4_PV := "DB_PLC1_MB_Buffer_DB".Recv_PID_Bon4_PV;
   END_IF;
END_REGION

REGION Network 83: Modbus TCP Client - Copy Recv PID_Bon4_CV
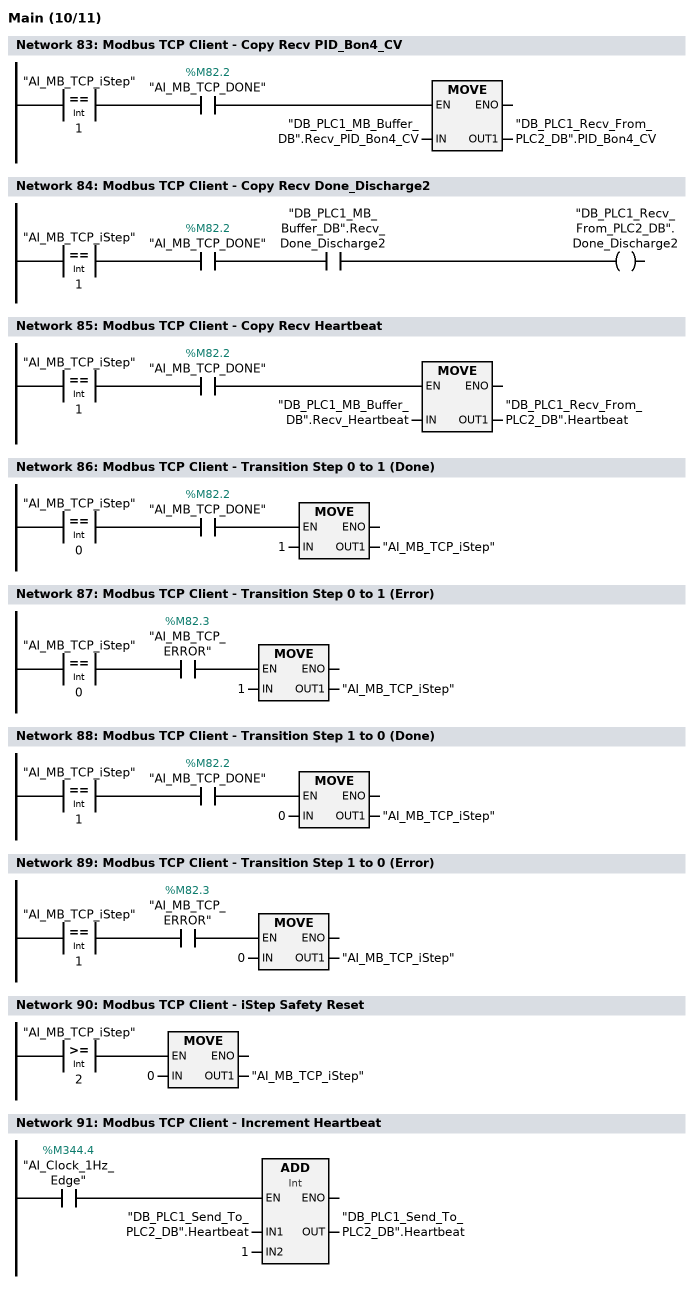
   RUNG wire#powerrail
      { S7_Templates := "SrcType := Int" } EQ_Contact(in1 := "AI_MB_TCP_iStep", in2 := 1)
      Contact( "AI_MB_TCP_DONE" )
      { S7_GenerateENO := "TRUE" } Move(in := "DB_PLC1_MB_Buffer_DB".Recv_PID_Bon4_CV, out1 => "DB_PLC1_Recv_From_PLC2_DB".PID_Bon4_CV)
   END_RUNG
   // the same network as SCL:
   IF ("AI_MB_TCP_iStep" = 1) AND "AI_MB_TCP_DONE" THEN
       "DB_PLC1_Recv_From_PLC2_DB".PID_Bon4_CV := "DB_PLC1_MB_Buffer_DB".Recv_PID_Bon4_CV;
   END_IF;
END_REGION

REGION Network 84: Modbus TCP Client - Copy Recv Done_Discharge2
   RUNG wire#powerrail
      { S7_Templates := "SrcType := Int" } EQ_Contact(in1 := "AI_MB_TCP_iStep", in2 := 1)
      Contact( "AI_MB_TCP_DONE" )
      Contact( "DB_PLC1_MB_Buffer_DB".Recv_Done_Discharge2 )
      Coil( "DB_PLC1_Recv_From_PLC2_DB".Done_Discharge2 )
   END_RUNG
   // the same network as SCL:
   "DB_PLC1_Recv_From_PLC2_DB".Done_Discharge2 := ("AI_MB_TCP_iStep" = 1) AND "AI_MB_TCP_DONE" AND "DB_PLC1_MB_Buffer_DB".Recv_Done_Discharge2;
END_REGION

REGION Network 85: Modbus TCP Client - Copy Recv Heartbeat
   RUNG wire#powerrail
      { S7_Templates := "SrcType := Int" } EQ_Contact(in1 := "AI_MB_TCP_iStep", in2 := 1)
      Contact( "AI_MB_TCP_DONE" )
      { S7_GenerateENO := "TRUE" } Move(in := "DB_PLC1_MB_Buffer_DB".Recv_Heartbeat, out1 => "DB_PLC1_Recv_From_PLC2_DB".Heartbeat)
   END_RUNG
   // the same network as SCL:
   IF ("AI_MB_TCP_iStep" = 1) AND "AI_MB_TCP_DONE" THEN
       "DB_PLC1_Recv_From_PLC2_DB".Heartbeat := "DB_PLC1_MB_Buffer_DB".Recv_Heartbeat;
   END_IF;
END_REGION

REGION Network 86: Modbus TCP Client - Transition Step 0 to 1 (Done)
   RUNG wire#powerrail
      { S7_Templates := "SrcType := Int" } EQ_Contact(in1 := "AI_MB_TCP_iStep", in2 := 0)
      Contact( "AI_MB_TCP_DONE" )
      { S7_GenerateENO := "TRUE" } Move(in := 1, out1 => "AI_MB_TCP_iStep")
   END_RUNG
   // the same network as SCL:
   IF ("AI_MB_TCP_iStep" = 0) AND "AI_MB_TCP_DONE" THEN "AI_MB_TCP_iStep" := 1; END_IF;
END_REGION

REGION Network 87: Modbus TCP Client - Transition Step 0 to 1 (Error)
   RUNG wire#powerrail
      { S7_Templates := "SrcType := Int" } EQ_Contact(in1 := "AI_MB_TCP_iStep", in2 := 0)
      Contact( "AI_MB_TCP_ERROR" )
      { S7_GenerateENO := "TRUE" } Move(in := 1, out1 => "AI_MB_TCP_iStep")
   END_RUNG
   // the same network as SCL:
   IF ("AI_MB_TCP_iStep" = 0) AND "AI_MB_TCP_ERROR" THEN "AI_MB_TCP_iStep" := 1; END_IF;
END_REGION

REGION Network 88: Modbus TCP Client - Transition Step 1 to 0 (Done)
   RUNG wire#powerrail
      { S7_Templates := "SrcType := Int" } EQ_Contact(in1 := "AI_MB_TCP_iStep", in2 := 1)
      Contact( "AI_MB_TCP_DONE" )
      { S7_GenerateENO := "TRUE" } Move(in := 0, out1 => "AI_MB_TCP_iStep")
   END_RUNG
   // the same network as SCL:
   IF ("AI_MB_TCP_iStep" = 1) AND "AI_MB_TCP_DONE" THEN "AI_MB_TCP_iStep" := 0; END_IF;
END_REGION

REGION Network 89: Modbus TCP Client - Transition Step 1 to 0 (Error)
   RUNG wire#powerrail
      { S7_Templates := "SrcType := Int" } EQ_Contact(in1 := "AI_MB_TCP_iStep", in2 := 1)
      Contact( "AI_MB_TCP_ERROR" )
      { S7_GenerateENO := "TRUE" } Move(in := 0, out1 => "AI_MB_TCP_iStep")
   END_RUNG
   // the same network as SCL:
   IF ("AI_MB_TCP_iStep" = 1) AND "AI_MB_TCP_ERROR" THEN "AI_MB_TCP_iStep" := 0; END_IF;
END_REGION

REGION Network 90: Modbus TCP Client - iStep Safety Reset
   RUNG wire#powerrail
      { S7_Templates := "SrcType := Int" } GE_Contact(in1 := "AI_MB_TCP_iStep", in2 := 2)
      { S7_GenerateENO := "TRUE" } Move(in := 0, out1 => "AI_MB_TCP_iStep")
   END_RUNG
   // the same network as SCL:
   IF "AI_MB_TCP_iStep" >= 2 THEN "AI_MB_TCP_iStep" := 0; END_IF;
END_REGION

REGION Network 91: Modbus TCP Client - Increment Heartbeat
   RUNG wire#powerrail
      Contact( "AI_Clock_1Hz_Edge" )
      { S7_Templates := "SrcType := Int"; S7_GenerateENO := "TRUE" } Add(in1 := "DB_PLC1_Send_To_PLC2_DB".Heartbeat, in2 := 1, out => "DB_PLC1_Send_To_PLC2_DB".Heartbeat)
   END_RUNG
   // the same network as SCL:
   IF "AI_Clock_1Hz_Edge" THEN
       "DB_PLC1_Send_To_PLC2_DB".Heartbeat := "DB_PLC1_Send_To_PLC2_DB".Heartbeat + 1;
   END_IF;
END_REGION

REGION Network 92: Modbus TCP Client - Monitor Heartbeat Change
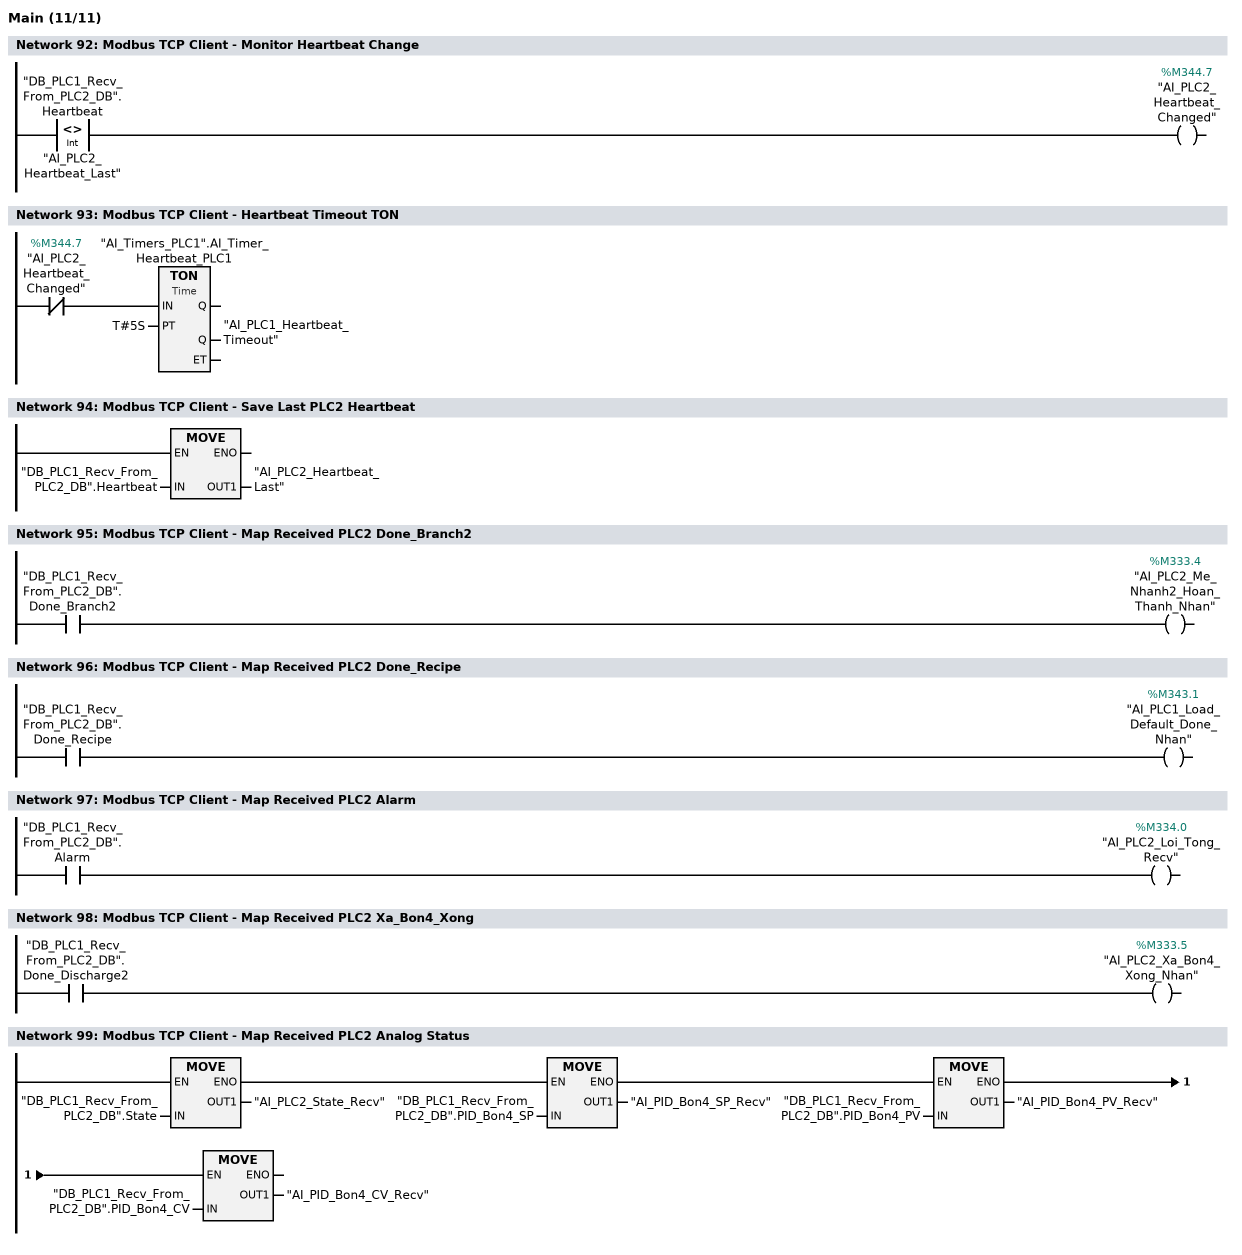
   RUNG wire#powerrail
      { S7_Templates := "SrcType := Int" } NE_Contact(in1 := "DB_PLC1_Recv_From_PLC2_DB".Heartbeat, in2 := "AI_PLC2_Heartbeat_Last")
      Coil( "AI_PLC2_Heartbeat_Changed" )
   END_RUNG
   // the same network as SCL:
   "AI_PLC2_Heartbeat_Changed" := "DB_PLC1_Recv_From_PLC2_DB".Heartbeat <> "AI_PLC2_Heartbeat_Last";
END_REGION

REGION Network 93: Modbus TCP Client - Heartbeat Timeout TON
   RUNG wire#powerrail
      I_Contact( "AI_PLC2_Heartbeat_Changed" )
      { S7_Templates := "time_type := Time" } "AI_Timers_PLC1".AI_Timer_Heartbeat_PLC1.TON(pt := T#5S, q => "AI_PLC1_Heartbeat_Timeout", et =>)
   END_RUNG
   // the same network as SCL:
   "AI_Timers_PLC1".AI_Timer_Heartbeat_PLC1.TON(IN := NOT "AI_PLC2_Heartbeat_Changed",
                           PT := T#5S,
                           Q => "AI_PLC1_Heartbeat_Timeout");
END_REGION

REGION Network 94: Modbus TCP Client - Save Last PLC2 Heartbeat
   RUNG wire#powerrail
      { S7_GenerateENO := "TRUE" } Move(in := "DB_PLC1_Recv_From_PLC2_DB".Heartbeat, out1 => "AI_PLC2_Heartbeat_Last")
   END_RUNG
   // the same network as SCL:
   "AI_PLC2_Heartbeat_Last" := "DB_PLC1_Recv_From_PLC2_DB".Heartbeat;
END_REGION

REGION Network 95: Modbus TCP Client - Map Received PLC2 Done_Branch2
   RUNG wire#powerrail
      Contact( "DB_PLC1_Recv_From_PLC2_DB".Done_Branch2 )
      Coil( "AI_PLC2_Me_Nhanh2_Hoan_Thanh_Nhan" )
   END_RUNG
   // the same network as SCL:
   "AI_PLC2_Me_Nhanh2_Hoan_Thanh_Nhan" := "DB_PLC1_Recv_From_PLC2_DB".Done_Branch2;
END_REGION

REGION Network 96: Modbus TCP Client - Map Received PLC2 Done_Recipe
   RUNG wire#powerrail
      Contact( "DB_PLC1_Recv_From_PLC2_DB".Done_Recipe )
      Coil( "AI_PLC1_Load_Default_Done_Nhan" )
   END_RUNG
   // the same network as SCL:
   "AI_PLC1_Load_Default_Done_Nhan" := "DB_PLC1_Recv_From_PLC2_DB".Done_Recipe;
END_REGION

REGION Network 97: Modbus TCP Client - Map Received PLC2 Alarm
   RUNG wire#powerrail
      Contact( "DB_PLC1_Recv_From_PLC2_DB".Alarm )
      Coil( "AI_PLC2_Loi_Tong_Recv" )
   END_RUNG
   // the same network as SCL:
   "AI_PLC2_Loi_Tong_Recv" := "DB_PLC1_Recv_From_PLC2_DB".Alarm;
END_REGION

REGION Network 98: Modbus TCP Client - Map Received PLC2 Xa_Bon4_Xong
   RUNG wire#powerrail
      Contact( "DB_PLC1_Recv_From_PLC2_DB".Done_Discharge2 )
      Coil( "AI_PLC2_Xa_Bon4_Xong_Nhan" )
   END_RUNG
   // the same network as SCL:
   "AI_PLC2_Xa_Bon4_Xong_Nhan" := "DB_PLC1_Recv_From_PLC2_DB".Done_Discharge2;
END_REGION

REGION Network 99: Modbus TCP Client - Map Received PLC2 Analog Status
   RUNG wire#powerrail
      { S7_GenerateENO := "TRUE" } Move(in := "DB_PLC1_Recv_From_PLC2_DB".State, out1 => "AI_PLC2_State_Recv")
      { S7_GenerateENO := "TRUE" } Move(in := "DB_PLC1_Recv_From_PLC2_DB".PID_Bon4_SP, out1 => "AI_PID_Bon4_SP_Recv")
      { S7_GenerateENO := "TRUE" } Move(in := "DB_PLC1_Recv_From_PLC2_DB".PID_Bon4_PV, out1 => "AI_PID_Bon4_PV_Recv")
      { S7_GenerateENO := "TRUE" } Move(in := "DB_PLC1_Recv_From_PLC2_DB".PID_Bon4_CV, out1 => "AI_PID_Bon4_CV_Recv")
   END_RUNG
   // the same network as SCL:
   // ENO of a box is taken as its EN; it also drops when the box reports an error
   "AI_PLC2_State_Recv" := "DB_PLC1_Recv_From_PLC2_DB".State;
   "AI_PID_Bon4_SP_Recv" := "DB_PLC1_Recv_From_PLC2_DB".PID_Bon4_SP;
   "AI_PID_Bon4_PV_Recv" := "DB_PLC1_Recv_From_PLC2_DB".PID_Bon4_PV;
   "AI_PID_Bon4_CV_Recv" := "DB_PLC1_Recv_From_PLC2_DB".PID_Bon4_CV;
END_REGION
END_ORGANIZATION_BLOCK

FUNCTION "FC_Init_Default_Recipe_PLC1" : Void   // FC50, LAD
{ S7_Optimized_Access := 'TRUE' }
VERSION : 0.1
// stored: AutoNumber true, IsIECCheckEnabled false
BEGIN

REGION Network 1: Kích hoạt nạp recipe mặc định lần đầu scan PLC1
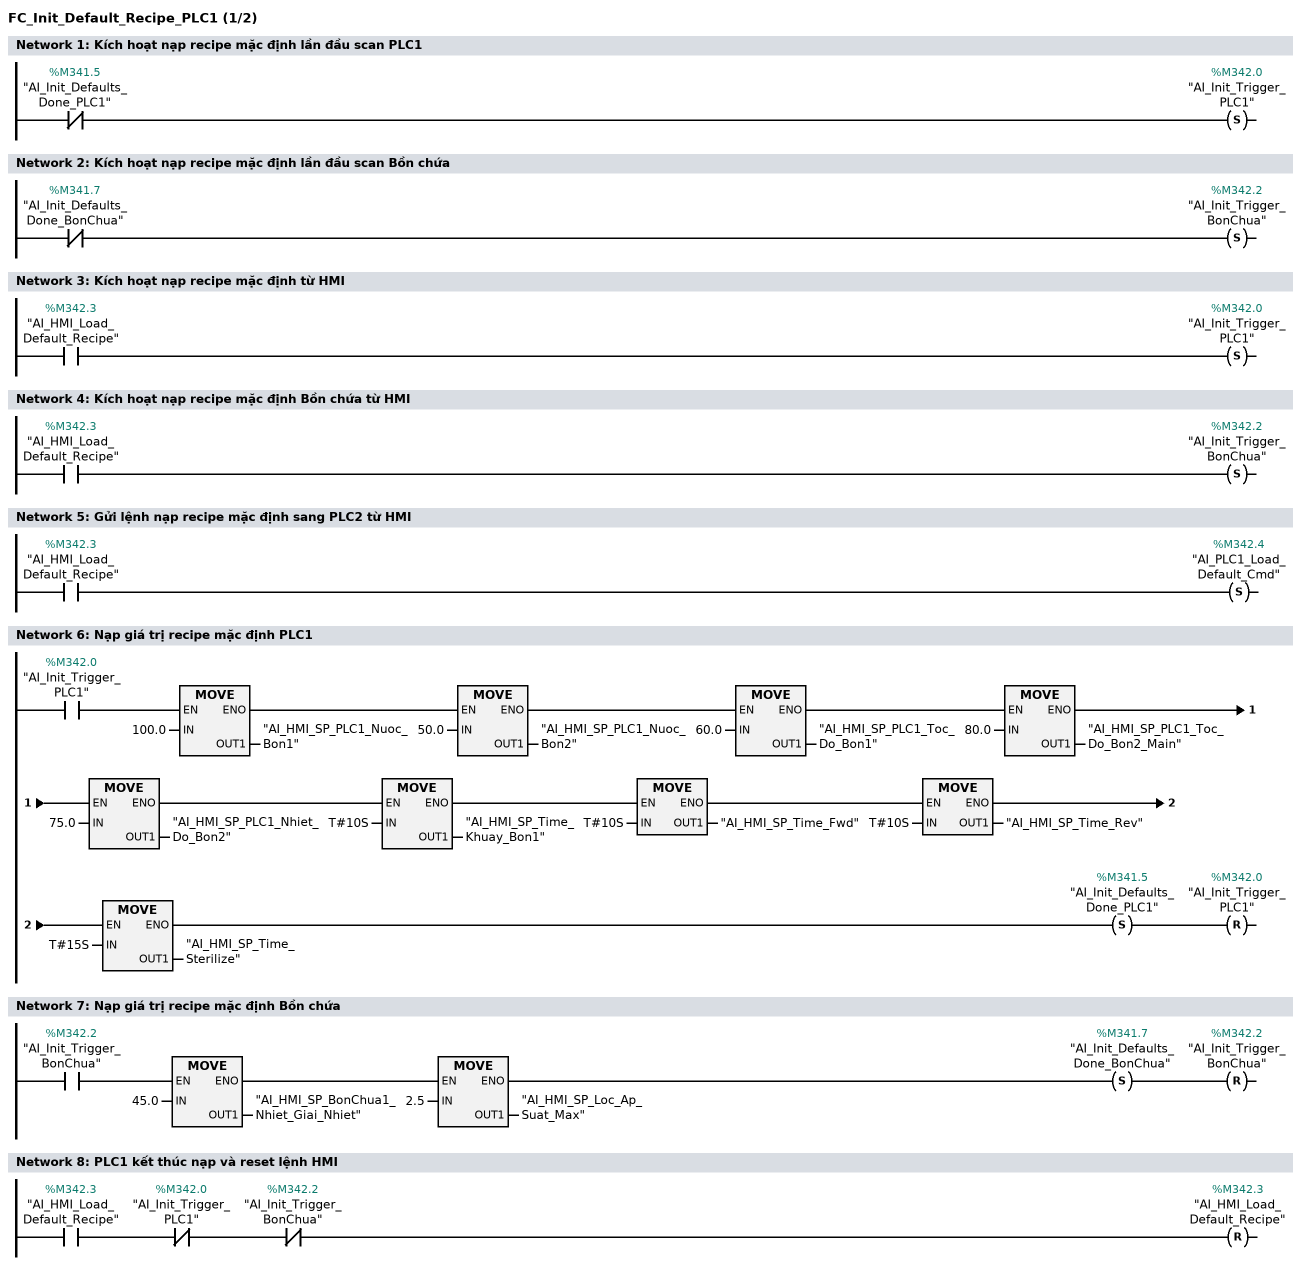
   RUNG wire#powerrail
      I_Contact( "AI_Init_Defaults_Done_PLC1" )
      S_Coil( "AI_Init_Trigger_PLC1" )
   END_RUNG
   // the same network as SCL:
   IF NOT "AI_Init_Defaults_Done_PLC1" THEN "AI_Init_Trigger_PLC1" := TRUE; END_IF;
END_REGION

REGION Network 2: Kích hoạt nạp recipe mặc định lần đầu scan Bồn chứa
   RUNG wire#powerrail
      I_Contact( "AI_Init_Defaults_Done_BonChua" )
      S_Coil( "AI_Init_Trigger_BonChua" )
   END_RUNG
   // the same network as SCL:
   IF NOT "AI_Init_Defaults_Done_BonChua" THEN "AI_Init_Trigger_BonChua" := TRUE; END_IF;
END_REGION

REGION Network 3: Kích hoạt nạp recipe mặc định từ HMI
   RUNG wire#powerrail
      Contact( "AI_HMI_Load_Default_Recipe" )
      S_Coil( "AI_Init_Trigger_PLC1" )
   END_RUNG
   // the same network as SCL:
   IF "AI_HMI_Load_Default_Recipe" THEN "AI_Init_Trigger_PLC1" := TRUE; END_IF;
END_REGION

REGION Network 4: Kích hoạt nạp recipe mặc định Bồn chứa từ HMI
   RUNG wire#powerrail
      Contact( "AI_HMI_Load_Default_Recipe" )
      S_Coil( "AI_Init_Trigger_BonChua" )
   END_RUNG
   // the same network as SCL:
   IF "AI_HMI_Load_Default_Recipe" THEN "AI_Init_Trigger_BonChua" := TRUE; END_IF;
END_REGION

REGION Network 5: Gửi lệnh nạp recipe mặc định sang PLC2 từ HMI
   RUNG wire#powerrail
      Contact( "AI_HMI_Load_Default_Recipe" )
      S_Coil( "AI_PLC1_Load_Default_Cmd" )
   END_RUNG
   // the same network as SCL:
   IF "AI_HMI_Load_Default_Recipe" THEN "AI_PLC1_Load_Default_Cmd" := TRUE; END_IF;
END_REGION

REGION Network 6: Nạp giá trị recipe mặc định PLC1
   RUNG wire#powerrail
      Contact( "AI_Init_Trigger_PLC1" )
      { S7_GenerateENO := "TRUE" } Move(in := 100.0, out1 => "AI_HMI_SP_PLC1_Nuoc_Bon1")
      { S7_GenerateENO := "TRUE" } Move(in := 50.0, out1 => "AI_HMI_SP_PLC1_Nuoc_Bon2")
      { S7_GenerateENO := "TRUE" } Move(in := 60.0, out1 => "AI_HMI_SP_PLC1_Toc_Do_Bon1")
      { S7_GenerateENO := "TRUE" } Move(in := 80.0, out1 => "AI_HMI_SP_PLC1_Toc_Do_Bon2_Main")
      { S7_GenerateENO := "TRUE" } Move(in := 75.0, out1 => "AI_HMI_SP_PLC1_Nhiet_Do_Bon2")
      { S7_GenerateENO := "TRUE" } Move(in := T#10S, out1 => "AI_HMI_SP_Time_Khuay_Bon1")
      { S7_GenerateENO := "TRUE" } Move(in := T#10S, out1 => "AI_HMI_SP_Time_Fwd")
      { S7_GenerateENO := "TRUE" } Move(in := T#10S, out1 => "AI_HMI_SP_Time_Rev")
      { S7_GenerateENO := "TRUE" } Move(in := T#15S, out1 => "AI_HMI_SP_Time_Sterilize")
      S_Coil( "AI_Init_Defaults_Done_PLC1" )
      R_Coil( "AI_Init_Trigger_PLC1" )
   END_RUNG
   // the same network as SCL:
   // ENO of a box is taken as its EN; it also drops when the box reports an error
   IF "AI_Init_Trigger_PLC1" THEN
       "AI_HMI_SP_PLC1_Nuoc_Bon1" := 100.0;
       "AI_HMI_SP_PLC1_Nuoc_Bon2" := 50.0;
       "AI_HMI_SP_PLC1_Toc_Do_Bon1" := 60.0;
       "AI_HMI_SP_PLC1_Toc_Do_Bon2_Main" := 80.0;
       "AI_HMI_SP_PLC1_Nhiet_Do_Bon2" := 75.0;
       "AI_HMI_SP_Time_Khuay_Bon1" := T#10S;
       "AI_HMI_SP_Time_Fwd" := T#10S;
       "AI_HMI_SP_Time_Rev" := T#10S;
       "AI_HMI_SP_Time_Sterilize" := T#15S;
       "AI_Init_Defaults_Done_PLC1" := TRUE;
       "AI_Init_Trigger_PLC1" := FALSE;
   END_IF;
END_REGION

REGION Network 7: Nạp giá trị recipe mặc định Bồn chứa
   RUNG wire#powerrail
      Contact( "AI_Init_Trigger_BonChua" )
      { S7_GenerateENO := "TRUE" } Move(in := 45.0, out1 => "AI_HMI_SP_BonChua1_Nhiet_Giai_Nhiet")
      { S7_GenerateENO := "TRUE" } Move(in := 2.5, out1 => "AI_HMI_SP_Loc_Ap_Suat_Max")
      S_Coil( "AI_Init_Defaults_Done_BonChua" )
      R_Coil( "AI_Init_Trigger_BonChua" )
   END_RUNG
   // the same network as SCL:
   // ENO of a box is taken as its EN; it also drops when the box reports an error
   IF "AI_Init_Trigger_BonChua" THEN
       "AI_HMI_SP_BonChua1_Nhiet_Giai_Nhiet" := 45.0;
       "AI_HMI_SP_Loc_Ap_Suat_Max" := 2.5;
       "AI_Init_Defaults_Done_BonChua" := TRUE;
       "AI_Init_Trigger_BonChua" := FALSE;
   END_IF;
END_REGION

REGION Network 8: PLC1 kết thúc nạp và reset lệnh HMI
   RUNG wire#powerrail
      Contact( "AI_HMI_Load_Default_Recipe" )
      I_Contact( "AI_Init_Trigger_PLC1" )
      I_Contact( "AI_Init_Trigger_BonChua" )
      R_Coil( "AI_HMI_Load_Default_Recipe" )
   END_RUNG
   // the same network as SCL:
   IF "AI_HMI_Load_Default_Recipe" AND NOT "AI_Init_Trigger_PLC1" AND NOT "AI_Init_Trigger_BonChua" THEN
       "AI_HMI_Load_Default_Recipe" := FALSE;
   END_IF;
END_REGION

REGION Network 9: PLC1 reset lệnh truyền thông nạp mặc định
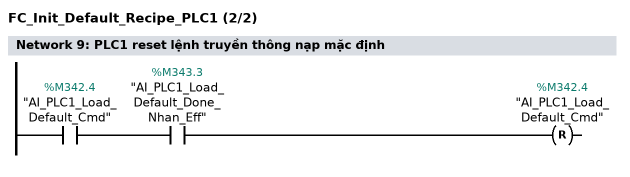
   RUNG wire#powerrail
      Contact( "AI_PLC1_Load_Default_Cmd" )
      Contact( "AI_PLC1_Load_Default_Done_Nhan_Eff" )
      R_Coil( "AI_PLC1_Load_Default_Cmd" )
   END_RUNG
   // the same network as SCL:
   IF "AI_PLC1_Load_Default_Cmd" AND "AI_PLC1_Load_Default_Done_Nhan_Eff" THEN
       "AI_PLC1_Load_Default_Cmd" := FALSE;
   END_IF;
END_REGION
END_FUNCTION

FUNCTION "FC_PLC1_Mixing" : Void   // FC10, LAD
{ S7_Optimized_Access := 'TRUE' }
VERSION : 0.1
// stored: AutoNumber true, IsIECCheckEnabled false
   VAR_TEMP   // added for the SCL form of the ladder/FBD networks
      _w1 : Bool;
   END_VAR
BEGIN

REGION Network 1: Khóa nút nhấn Start HMI qua Run Enable
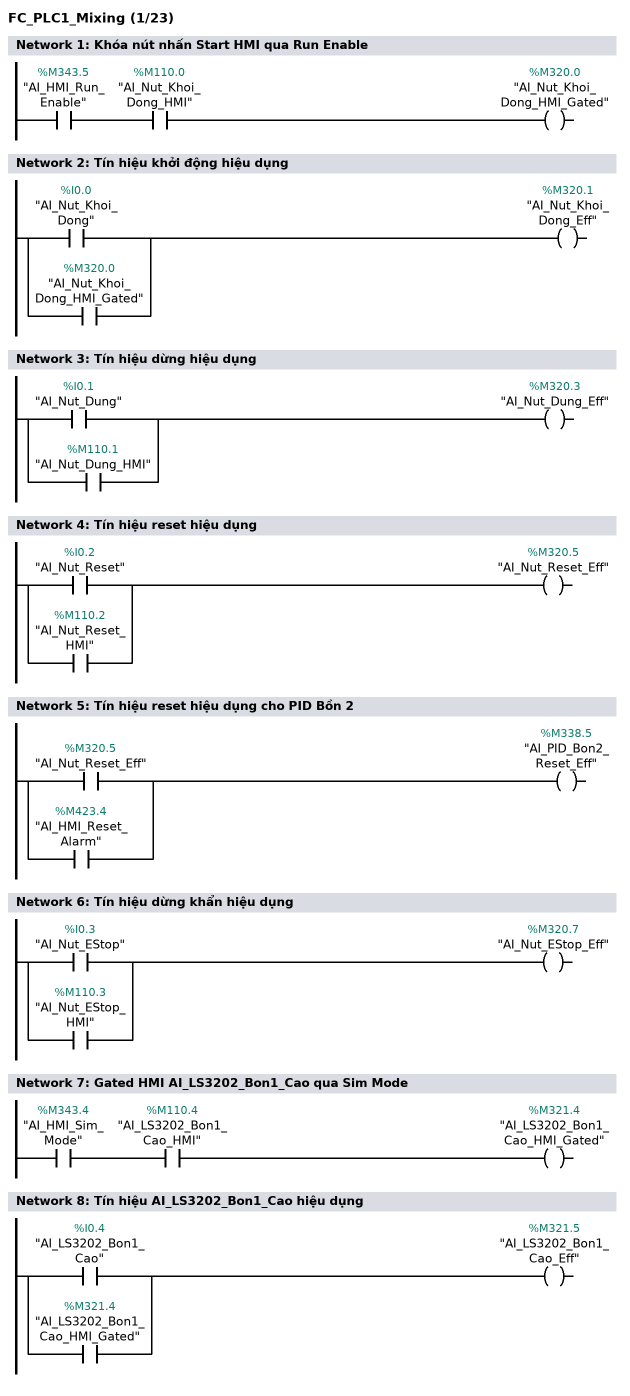
   RUNG wire#powerrail
      Contact( "AI_HMI_Run_Enable" )
      Contact( "AI_Nut_Khoi_Dong_HMI" )
      Coil( "AI_Nut_Khoi_Dong_HMI_Gated" )
   END_RUNG
   // the same network as SCL:
   "AI_Nut_Khoi_Dong_HMI_Gated" := "AI_HMI_Run_Enable" AND "AI_Nut_Khoi_Dong_HMI";
END_REGION

REGION Network 2: Tín hiệu khởi động hiệu dụng
   RUNG wire#powerrail
      Contact( "AI_Nut_Khoi_Dong" )
      wire#w1
      Coil( "AI_Nut_Khoi_Dong_Eff" )
   END_RUNG
   RUNG wire#powerrail
      Contact( "AI_Nut_Khoi_Dong_HMI_Gated" )
   END_RUNG wire#w1
   // the same network as SCL:
   "AI_Nut_Khoi_Dong_Eff" := "AI_Nut_Khoi_Dong" OR "AI_Nut_Khoi_Dong_HMI_Gated";
END_REGION

REGION Network 3: Tín hiệu dừng hiệu dụng
   RUNG wire#powerrail
      Contact( "AI_Nut_Dung" )
      wire#w1
      Coil( "AI_Nut_Dung_Eff" )
   END_RUNG
   RUNG wire#powerrail
      Contact( "AI_Nut_Dung_HMI" )
   END_RUNG wire#w1
   // the same network as SCL:
   "AI_Nut_Dung_Eff" := "AI_Nut_Dung" OR "AI_Nut_Dung_HMI";
END_REGION

REGION Network 4: Tín hiệu reset hiệu dụng
   RUNG wire#powerrail
      Contact( "AI_Nut_Reset" )
      wire#w1
      Coil( "AI_Nut_Reset_Eff" )
   END_RUNG
   RUNG wire#powerrail
      Contact( "AI_Nut_Reset_HMI" )
   END_RUNG wire#w1
   // the same network as SCL:
   "AI_Nut_Reset_Eff" := "AI_Nut_Reset" OR "AI_Nut_Reset_HMI";
END_REGION

REGION Network 5: Tín hiệu reset hiệu dụng cho PID Bồn 2
   RUNG wire#powerrail
      Contact( "AI_Nut_Reset_Eff" )
      wire#w1
      Coil( "AI_PID_Bon2_Reset_Eff" )
   END_RUNG
   RUNG wire#powerrail
      Contact( "AI_HMI_Reset_Alarm" )
   END_RUNG wire#w1
   // the same network as SCL:
   "AI_PID_Bon2_Reset_Eff" := "AI_Nut_Reset_Eff" OR "AI_HMI_Reset_Alarm";
END_REGION

REGION Network 6: Tín hiệu dừng khẩn hiệu dụng
   RUNG wire#powerrail
      Contact( "AI_Nut_EStop" )
      wire#w1
      Coil( "AI_Nut_EStop_Eff" )
   END_RUNG
   RUNG wire#powerrail
      Contact( "AI_Nut_EStop_HMI" )
   END_RUNG wire#w1
   // the same network as SCL:
   "AI_Nut_EStop_Eff" := "AI_Nut_EStop" OR "AI_Nut_EStop_HMI";
END_REGION

REGION Network 7: Gated HMI AI_LS3202_Bon1_Cao qua Sim Mode
   RUNG wire#powerrail
      Contact( "AI_HMI_Sim_Mode" )
      Contact( "AI_LS3202_Bon1_Cao_HMI" )
      Coil( "AI_LS3202_Bon1_Cao_HMI_Gated" )
   END_RUNG
   // the same network as SCL:
   "AI_LS3202_Bon1_Cao_HMI_Gated" := "AI_HMI_Sim_Mode" AND "AI_LS3202_Bon1_Cao_HMI";
END_REGION

REGION Network 8: Tín hiệu AI_LS3202_Bon1_Cao hiệu dụng
   RUNG wire#powerrail
      Contact( "AI_LS3202_Bon1_Cao" )
      wire#w1
      Coil( "AI_LS3202_Bon1_Cao_Eff" )
   END_RUNG
   RUNG wire#powerrail
      Contact( "AI_LS3202_Bon1_Cao_HMI_Gated" )
   END_RUNG wire#w1
   // the same network as SCL:
   "AI_LS3202_Bon1_Cao_Eff" := "AI_LS3202_Bon1_Cao" OR "AI_LS3202_Bon1_Cao_HMI_Gated";
END_REGION

REGION Network 9: Gated HMI AI_PLC2_Me_Nhanh2_Hoan_Thanh_Nhan qua Sim Mode
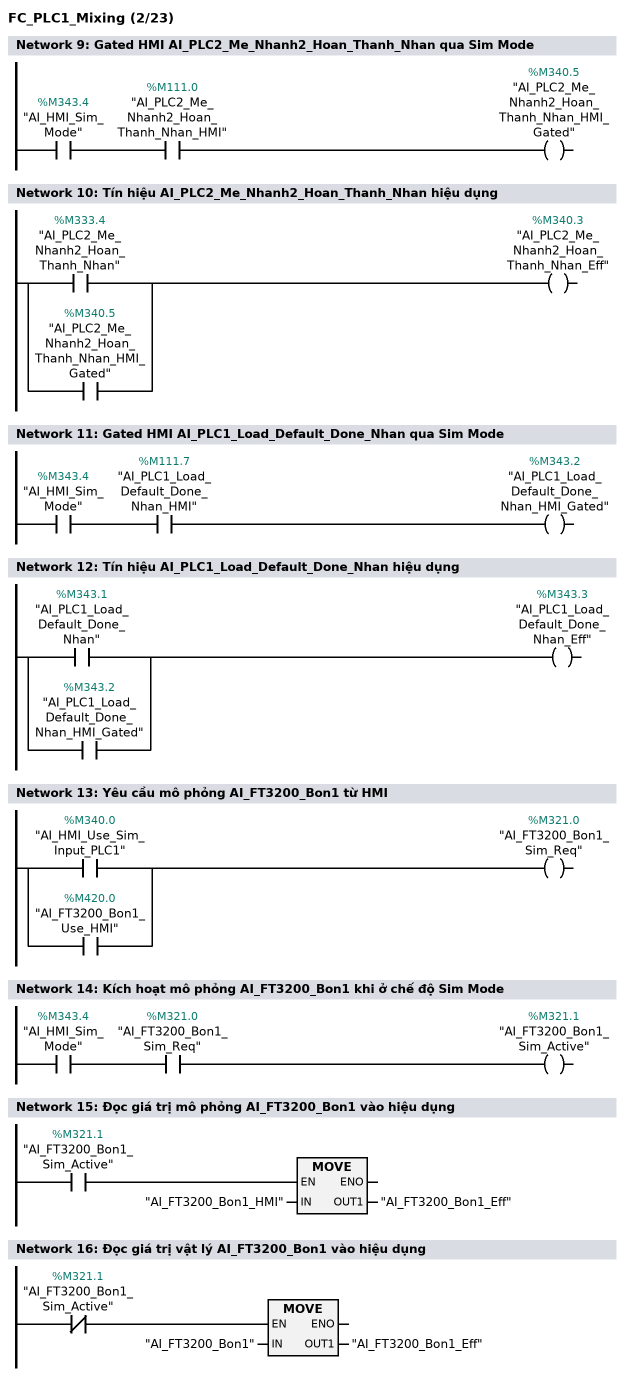
   RUNG wire#powerrail
      Contact( "AI_HMI_Sim_Mode" )
      Contact( "AI_PLC2_Me_Nhanh2_Hoan_Thanh_Nhan_HMI" )
      Coil( "AI_PLC2_Me_Nhanh2_Hoan_Thanh_Nhan_HMI_Gated" )
   END_RUNG
   // the same network as SCL:
   "AI_PLC2_Me_Nhanh2_Hoan_Thanh_Nhan_HMI_Gated" := "AI_HMI_Sim_Mode" AND "AI_PLC2_Me_Nhanh2_Hoan_Thanh_Nhan_HMI";
END_REGION

REGION Network 10: Tín hiệu AI_PLC2_Me_Nhanh2_Hoan_Thanh_Nhan hiệu dụng
   RUNG wire#powerrail
      Contact( "AI_PLC2_Me_Nhanh2_Hoan_Thanh_Nhan" )
      wire#w1
      Coil( "AI_PLC2_Me_Nhanh2_Hoan_Thanh_Nhan_Eff" )
   END_RUNG
   RUNG wire#powerrail
      Contact( "AI_PLC2_Me_Nhanh2_Hoan_Thanh_Nhan_HMI_Gated" )
   END_RUNG wire#w1
   // the same network as SCL:
   "AI_PLC2_Me_Nhanh2_Hoan_Thanh_Nhan_Eff" := "AI_PLC2_Me_Nhanh2_Hoan_Thanh_Nhan" OR "AI_PLC2_Me_Nhanh2_Hoan_Thanh_Nhan_HMI_Gated";
END_REGION

REGION Network 11: Gated HMI AI_PLC1_Load_Default_Done_Nhan qua Sim Mode
   RUNG wire#powerrail
      Contact( "AI_HMI_Sim_Mode" )
      Contact( "AI_PLC1_Load_Default_Done_Nhan_HMI" )
      Coil( "AI_PLC1_Load_Default_Done_Nhan_HMI_Gated" )
   END_RUNG
   // the same network as SCL:
   "AI_PLC1_Load_Default_Done_Nhan_HMI_Gated" := "AI_HMI_Sim_Mode" AND "AI_PLC1_Load_Default_Done_Nhan_HMI";
END_REGION

REGION Network 12: Tín hiệu AI_PLC1_Load_Default_Done_Nhan hiệu dụng
   RUNG wire#powerrail
      Contact( "AI_PLC1_Load_Default_Done_Nhan" )
      wire#w1
      Coil( "AI_PLC1_Load_Default_Done_Nhan_Eff" )
   END_RUNG
   RUNG wire#powerrail
      Contact( "AI_PLC1_Load_Default_Done_Nhan_HMI_Gated" )
   END_RUNG wire#w1
   // the same network as SCL:
   "AI_PLC1_Load_Default_Done_Nhan_Eff" := "AI_PLC1_Load_Default_Done_Nhan" OR "AI_PLC1_Load_Default_Done_Nhan_HMI_Gated";
END_REGION

REGION Network 13: Yêu cầu mô phỏng AI_FT3200_Bon1 từ HMI
   RUNG wire#powerrail
      Contact( "AI_HMI_Use_Sim_Input_PLC1" )
      wire#w1
      Coil( "AI_FT3200_Bon1_Sim_Req" )
   END_RUNG
   RUNG wire#powerrail
      Contact( "AI_FT3200_Bon1_Use_HMI" )
   END_RUNG wire#w1
   // the same network as SCL:
   "AI_FT3200_Bon1_Sim_Req" := "AI_HMI_Use_Sim_Input_PLC1" OR "AI_FT3200_Bon1_Use_HMI";
END_REGION

REGION Network 14: Kích hoạt mô phỏng AI_FT3200_Bon1 khi ở chế độ Sim Mode
   RUNG wire#powerrail
      Contact( "AI_HMI_Sim_Mode" )
      Contact( "AI_FT3200_Bon1_Sim_Req" )
      Coil( "AI_FT3200_Bon1_Sim_Active" )
   END_RUNG
   // the same network as SCL:
   "AI_FT3200_Bon1_Sim_Active" := "AI_HMI_Sim_Mode" AND "AI_FT3200_Bon1_Sim_Req";
END_REGION

REGION Network 15: Đọc giá trị mô phỏng AI_FT3200_Bon1 vào hiệu dụng
   RUNG wire#powerrail
      Contact( "AI_FT3200_Bon1_Sim_Active" )
      { S7_GenerateENO := "TRUE" } Move(in := "AI_FT3200_Bon1_HMI", out1 => "AI_FT3200_Bon1_Eff")
   END_RUNG
   // the same network as SCL:
   IF "AI_FT3200_Bon1_Sim_Active" THEN "AI_FT3200_Bon1_Eff" := "AI_FT3200_Bon1_HMI"; END_IF;
END_REGION

REGION Network 16: Đọc giá trị vật lý AI_FT3200_Bon1 vào hiệu dụng
   RUNG wire#powerrail
      I_Contact( "AI_FT3200_Bon1_Sim_Active" )
      { S7_GenerateENO := "TRUE" } Move(in := "AI_FT3200_Bon1", out1 => "AI_FT3200_Bon1_Eff")
   END_RUNG
   // the same network as SCL:
   IF NOT "AI_FT3200_Bon1_Sim_Active" THEN "AI_FT3200_Bon1_Eff" := "AI_FT3200_Bon1"; END_IF;
END_REGION

REGION Network 17: Yêu cầu mô phỏng AI_FQ3200_Bon1 từ HMI
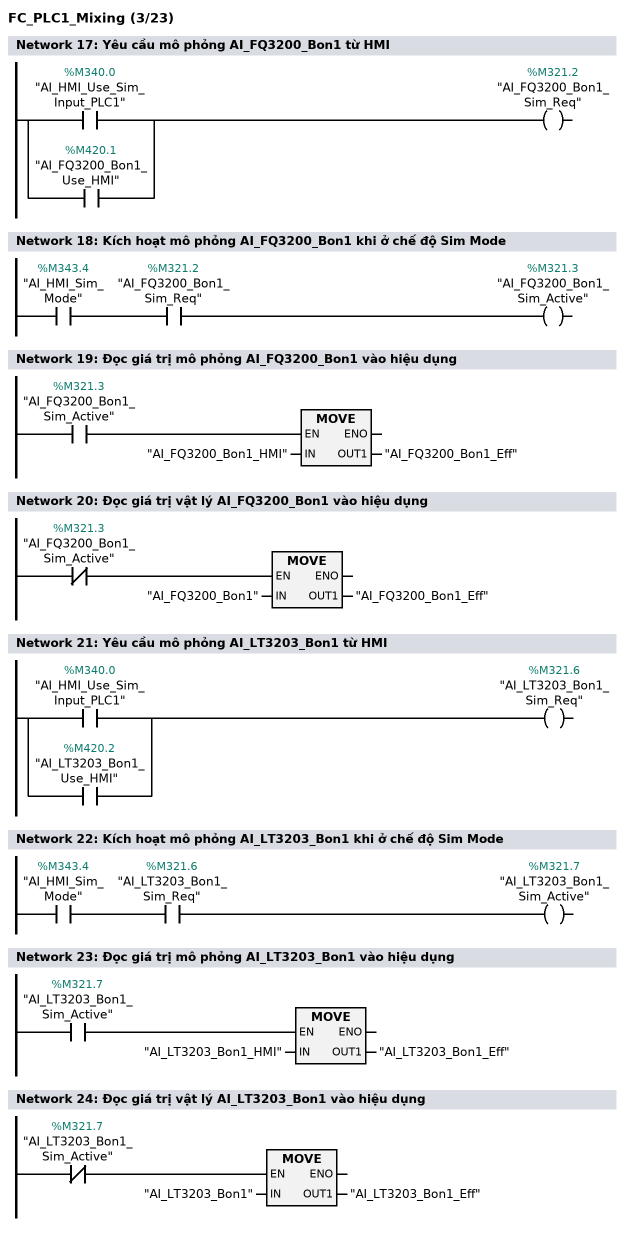
   RUNG wire#powerrail
      Contact( "AI_HMI_Use_Sim_Input_PLC1" )
      wire#w1
      Coil( "AI_FQ3200_Bon1_Sim_Req" )
   END_RUNG
   RUNG wire#powerrail
      Contact( "AI_FQ3200_Bon1_Use_HMI" )
   END_RUNG wire#w1
   // the same network as SCL:
   "AI_FQ3200_Bon1_Sim_Req" := "AI_HMI_Use_Sim_Input_PLC1" OR "AI_FQ3200_Bon1_Use_HMI";
END_REGION

REGION Network 18: Kích hoạt mô phỏng AI_FQ3200_Bon1 khi ở chế độ Sim Mode
   RUNG wire#powerrail
      Contact( "AI_HMI_Sim_Mode" )
      Contact( "AI_FQ3200_Bon1_Sim_Req" )
      Coil( "AI_FQ3200_Bon1_Sim_Active" )
   END_RUNG
   // the same network as SCL:
   "AI_FQ3200_Bon1_Sim_Active" := "AI_HMI_Sim_Mode" AND "AI_FQ3200_Bon1_Sim_Req";
END_REGION

REGION Network 19: Đọc giá trị mô phỏng AI_FQ3200_Bon1 vào hiệu dụng
   RUNG wire#powerrail
      Contact( "AI_FQ3200_Bon1_Sim_Active" )
      { S7_GenerateENO := "TRUE" } Move(in := "AI_FQ3200_Bon1_HMI", out1 => "AI_FQ3200_Bon1_Eff")
   END_RUNG
   // the same network as SCL:
   IF "AI_FQ3200_Bon1_Sim_Active" THEN "AI_FQ3200_Bon1_Eff" := "AI_FQ3200_Bon1_HMI"; END_IF;
END_REGION

REGION Network 20: Đọc giá trị vật lý AI_FQ3200_Bon1 vào hiệu dụng
   RUNG wire#powerrail
      I_Contact( "AI_FQ3200_Bon1_Sim_Active" )
      { S7_GenerateENO := "TRUE" } Move(in := "AI_FQ3200_Bon1", out1 => "AI_FQ3200_Bon1_Eff")
   END_RUNG
   // the same network as SCL:
   IF NOT "AI_FQ3200_Bon1_Sim_Active" THEN "AI_FQ3200_Bon1_Eff" := "AI_FQ3200_Bon1"; END_IF;
END_REGION

REGION Network 21: Yêu cầu mô phỏng AI_LT3203_Bon1 từ HMI
   RUNG wire#powerrail
      Contact( "AI_HMI_Use_Sim_Input_PLC1" )
      wire#w1
      Coil( "AI_LT3203_Bon1_Sim_Req" )
   END_RUNG
   RUNG wire#powerrail
      Contact( "AI_LT3203_Bon1_Use_HMI" )
   END_RUNG wire#w1
   // the same network as SCL:
   "AI_LT3203_Bon1_Sim_Req" := "AI_HMI_Use_Sim_Input_PLC1" OR "AI_LT3203_Bon1_Use_HMI";
END_REGION

REGION Network 22: Kích hoạt mô phỏng AI_LT3203_Bon1 khi ở chế độ Sim Mode
   RUNG wire#powerrail
      Contact( "AI_HMI_Sim_Mode" )
      Contact( "AI_LT3203_Bon1_Sim_Req" )
      Coil( "AI_LT3203_Bon1_Sim_Active" )
   END_RUNG
   // the same network as SCL:
   "AI_LT3203_Bon1_Sim_Active" := "AI_HMI_Sim_Mode" AND "AI_LT3203_Bon1_Sim_Req";
END_REGION

REGION Network 23: Đọc giá trị mô phỏng AI_LT3203_Bon1 vào hiệu dụng
   RUNG wire#powerrail
      Contact( "AI_LT3203_Bon1_Sim_Active" )
      { S7_GenerateENO := "TRUE" } Move(in := "AI_LT3203_Bon1_HMI", out1 => "AI_LT3203_Bon1_Eff")
   END_RUNG
   // the same network as SCL:
   IF "AI_LT3203_Bon1_Sim_Active" THEN "AI_LT3203_Bon1_Eff" := "AI_LT3203_Bon1_HMI"; END_IF;
END_REGION

REGION Network 24: Đọc giá trị vật lý AI_LT3203_Bon1 vào hiệu dụng
   RUNG wire#powerrail
      I_Contact( "AI_LT3203_Bon1_Sim_Active" )
      { S7_GenerateENO := "TRUE" } Move(in := "AI_LT3203_Bon1", out1 => "AI_LT3203_Bon1_Eff")
   END_RUNG
   // the same network as SCL:
   IF NOT "AI_LT3203_Bon1_Sim_Active" THEN "AI_LT3203_Bon1_Eff" := "AI_LT3203_Bon1"; END_IF;
END_REGION

REGION Network 25: Yêu cầu mô phỏng AI_TT3204_Bon1 từ HMI
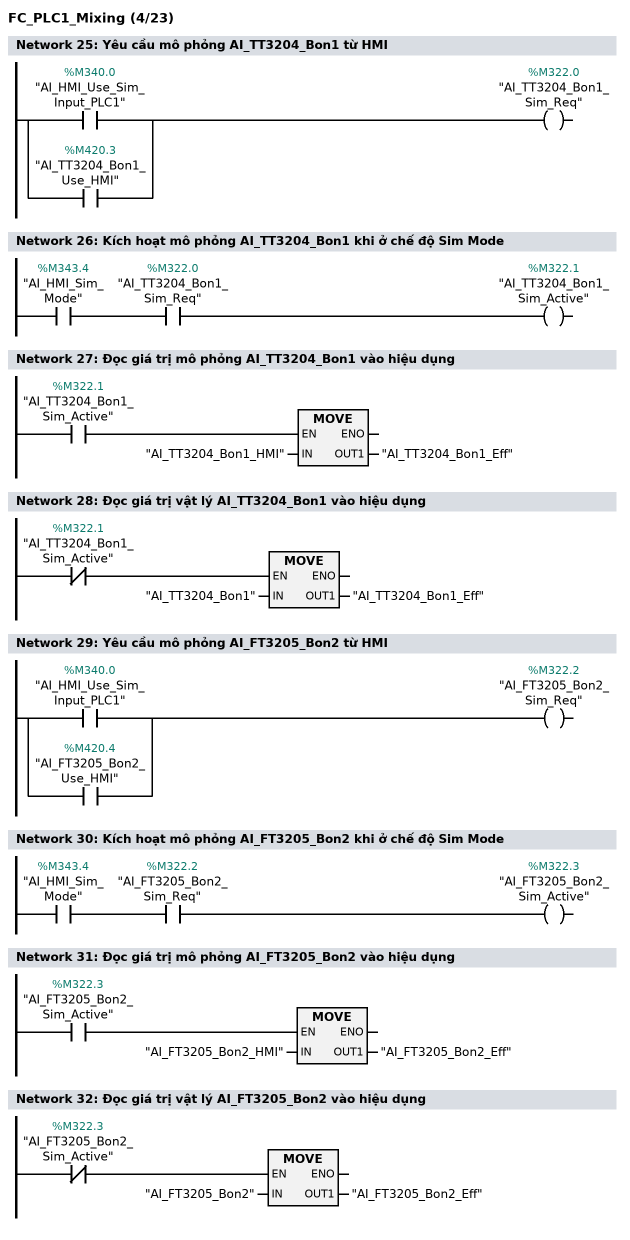
   RUNG wire#powerrail
      Contact( "AI_HMI_Use_Sim_Input_PLC1" )
      wire#w1
      Coil( "AI_TT3204_Bon1_Sim_Req" )
   END_RUNG
   RUNG wire#powerrail
      Contact( "AI_TT3204_Bon1_Use_HMI" )
   END_RUNG wire#w1
   // the same network as SCL:
   "AI_TT3204_Bon1_Sim_Req" := "AI_HMI_Use_Sim_Input_PLC1" OR "AI_TT3204_Bon1_Use_HMI";
END_REGION

REGION Network 26: Kích hoạt mô phỏng AI_TT3204_Bon1 khi ở chế độ Sim Mode
   RUNG wire#powerrail
      Contact( "AI_HMI_Sim_Mode" )
      Contact( "AI_TT3204_Bon1_Sim_Req" )
      Coil( "AI_TT3204_Bon1_Sim_Active" )
   END_RUNG
   // the same network as SCL:
   "AI_TT3204_Bon1_Sim_Active" := "AI_HMI_Sim_Mode" AND "AI_TT3204_Bon1_Sim_Req";
END_REGION

REGION Network 27: Đọc giá trị mô phỏng AI_TT3204_Bon1 vào hiệu dụng
   RUNG wire#powerrail
      Contact( "AI_TT3204_Bon1_Sim_Active" )
      { S7_GenerateENO := "TRUE" } Move(in := "AI_TT3204_Bon1_HMI", out1 => "AI_TT3204_Bon1_Eff")
   END_RUNG
   // the same network as SCL:
   IF "AI_TT3204_Bon1_Sim_Active" THEN "AI_TT3204_Bon1_Eff" := "AI_TT3204_Bon1_HMI"; END_IF;
END_REGION

REGION Network 28: Đọc giá trị vật lý AI_TT3204_Bon1 vào hiệu dụng
   RUNG wire#powerrail
      I_Contact( "AI_TT3204_Bon1_Sim_Active" )
      { S7_GenerateENO := "TRUE" } Move(in := "AI_TT3204_Bon1", out1 => "AI_TT3204_Bon1_Eff")
   END_RUNG
   // the same network as SCL:
   IF NOT "AI_TT3204_Bon1_Sim_Active" THEN "AI_TT3204_Bon1_Eff" := "AI_TT3204_Bon1"; END_IF;
END_REGION

REGION Network 29: Yêu cầu mô phỏng AI_FT3205_Bon2 từ HMI
   RUNG wire#powerrail
      Contact( "AI_HMI_Use_Sim_Input_PLC1" )
      wire#w1
      Coil( "AI_FT3205_Bon2_Sim_Req" )
   END_RUNG
   RUNG wire#powerrail
      Contact( "AI_FT3205_Bon2_Use_HMI" )
   END_RUNG wire#w1
   // the same network as SCL:
   "AI_FT3205_Bon2_Sim_Req" := "AI_HMI_Use_Sim_Input_PLC1" OR "AI_FT3205_Bon2_Use_HMI";
END_REGION

REGION Network 30: Kích hoạt mô phỏng AI_FT3205_Bon2 khi ở chế độ Sim Mode
   RUNG wire#powerrail
      Contact( "AI_HMI_Sim_Mode" )
      Contact( "AI_FT3205_Bon2_Sim_Req" )
      Coil( "AI_FT3205_Bon2_Sim_Active" )
   END_RUNG
   // the same network as SCL:
   "AI_FT3205_Bon2_Sim_Active" := "AI_HMI_Sim_Mode" AND "AI_FT3205_Bon2_Sim_Req";
END_REGION

REGION Network 31: Đọc giá trị mô phỏng AI_FT3205_Bon2 vào hiệu dụng
   RUNG wire#powerrail
      Contact( "AI_FT3205_Bon2_Sim_Active" )
      { S7_GenerateENO := "TRUE" } Move(in := "AI_FT3205_Bon2_HMI", out1 => "AI_FT3205_Bon2_Eff")
   END_RUNG
   // the same network as SCL:
   IF "AI_FT3205_Bon2_Sim_Active" THEN "AI_FT3205_Bon2_Eff" := "AI_FT3205_Bon2_HMI"; END_IF;
END_REGION

REGION Network 32: Đọc giá trị vật lý AI_FT3205_Bon2 vào hiệu dụng
   RUNG wire#powerrail
      I_Contact( "AI_FT3205_Bon2_Sim_Active" )
      { S7_GenerateENO := "TRUE" } Move(in := "AI_FT3205_Bon2", out1 => "AI_FT3205_Bon2_Eff")
   END_RUNG
   // the same network as SCL:
   IF NOT "AI_FT3205_Bon2_Sim_Active" THEN "AI_FT3205_Bon2_Eff" := "AI_FT3205_Bon2"; END_IF;
END_REGION

REGION Network 33: Yêu cầu mô phỏng AI_FQ3205_Bon2 từ HMI
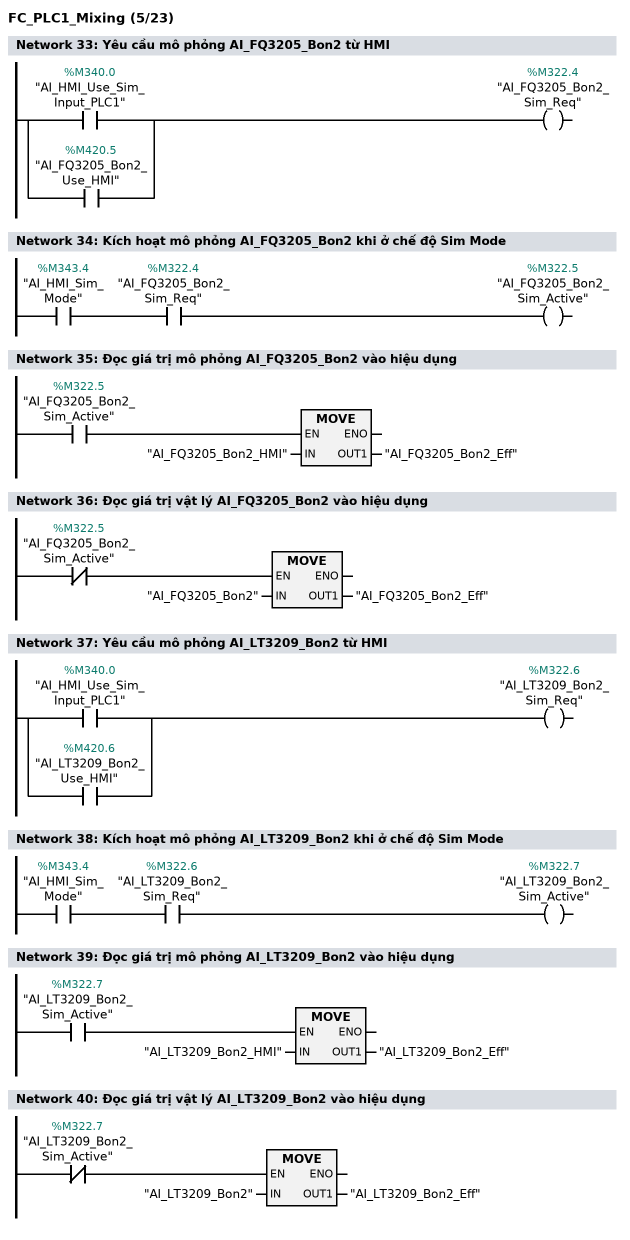
   RUNG wire#powerrail
      Contact( "AI_HMI_Use_Sim_Input_PLC1" )
      wire#w1
      Coil( "AI_FQ3205_Bon2_Sim_Req" )
   END_RUNG
   RUNG wire#powerrail
      Contact( "AI_FQ3205_Bon2_Use_HMI" )
   END_RUNG wire#w1
   // the same network as SCL:
   "AI_FQ3205_Bon2_Sim_Req" := "AI_HMI_Use_Sim_Input_PLC1" OR "AI_FQ3205_Bon2_Use_HMI";
END_REGION

REGION Network 34: Kích hoạt mô phỏng AI_FQ3205_Bon2 khi ở chế độ Sim Mode
   RUNG wire#powerrail
      Contact( "AI_HMI_Sim_Mode" )
      Contact( "AI_FQ3205_Bon2_Sim_Req" )
      Coil( "AI_FQ3205_Bon2_Sim_Active" )
   END_RUNG
   // the same network as SCL:
   "AI_FQ3205_Bon2_Sim_Active" := "AI_HMI_Sim_Mode" AND "AI_FQ3205_Bon2_Sim_Req";
END_REGION

REGION Network 35: Đọc giá trị mô phỏng AI_FQ3205_Bon2 vào hiệu dụng
   RUNG wire#powerrail
      Contact( "AI_FQ3205_Bon2_Sim_Active" )
      { S7_GenerateENO := "TRUE" } Move(in := "AI_FQ3205_Bon2_HMI", out1 => "AI_FQ3205_Bon2_Eff")
   END_RUNG
   // the same network as SCL:
   IF "AI_FQ3205_Bon2_Sim_Active" THEN "AI_FQ3205_Bon2_Eff" := "AI_FQ3205_Bon2_HMI"; END_IF;
END_REGION

REGION Network 36: Đọc giá trị vật lý AI_FQ3205_Bon2 vào hiệu dụng
   RUNG wire#powerrail
      I_Contact( "AI_FQ3205_Bon2_Sim_Active" )
      { S7_GenerateENO := "TRUE" } Move(in := "AI_FQ3205_Bon2", out1 => "AI_FQ3205_Bon2_Eff")
   END_RUNG
   // the same network as SCL:
   IF NOT "AI_FQ3205_Bon2_Sim_Active" THEN "AI_FQ3205_Bon2_Eff" := "AI_FQ3205_Bon2"; END_IF;
END_REGION

REGION Network 37: Yêu cầu mô phỏng AI_LT3209_Bon2 từ HMI
   RUNG wire#powerrail
      Contact( "AI_HMI_Use_Sim_Input_PLC1" )
      wire#w1
      Coil( "AI_LT3209_Bon2_Sim_Req" )
   END_RUNG
   RUNG wire#powerrail
      Contact( "AI_LT3209_Bon2_Use_HMI" )
   END_RUNG wire#w1
   // the same network as SCL:
   "AI_LT3209_Bon2_Sim_Req" := "AI_HMI_Use_Sim_Input_PLC1" OR "AI_LT3209_Bon2_Use_HMI";
END_REGION

REGION Network 38: Kích hoạt mô phỏng AI_LT3209_Bon2 khi ở chế độ Sim Mode
   RUNG wire#powerrail
      Contact( "AI_HMI_Sim_Mode" )
      Contact( "AI_LT3209_Bon2_Sim_Req" )
      Coil( "AI_LT3209_Bon2_Sim_Active" )
   END_RUNG
   // the same network as SCL:
   "AI_LT3209_Bon2_Sim_Active" := "AI_HMI_Sim_Mode" AND "AI_LT3209_Bon2_Sim_Req";
END_REGION

